The hash table can be thought of as an array on steriods, they are worth reading about, suffice to say
the hash table will tell you when you reach the end of all the entries, and enables us to find entries quickly.

These features efficiently address the addition, removal, and verification of beam parameter sets listed in the above requirements.
*)
{attribute 'reflection'}
FUNCTION_BLOCK FB_Arbiter IMPLEMENTS I_HigherAuthority, I_LowerAuthority
VAR
    nRequestsCount : UDINT; // How many requests are currently in the arbiter

    {attribute 'pytmc' := '
        pv: AP
        io: i
        field: DESC Assertion Pool
     '}
    fbBPAssertionPool    :    FB_BeamParamAssertionPool; //Table of active beam parameter assertions

    xRequestMade : BOOL; // Arbiter has confirmed its request has made it into the beam parameter request

    {attribute 'pytmc' := '
        pv: ArbiterID
        io: i
        field: DESC Arbiter ID for elev. req.
     '}
    nArbiterID : UDINT; // Arbiter ID, used for making higher-level BP requests

    nNextCohort : UDINT := 1; // The cohort ID any new requests will adopt, will become ReqInProgCohort at the start of the next acknowledgement cycle
    nAckInProgCohort : UDINT := 0; // The cohort ID currently being acknowledged, will become nActiveCohort after acknowledgement from HA
    {attribute 'pytmc' := '
        pv: CohortCounter
        io: i
        field: DESC Intrnl cohort counter
     '}
    nActiveCohort : UDINT := 0; // Requests with cohorts <= to this value will be considered active in CheckRequest

    bStartNewAckRequest : BOOL; // Set by an add or remove method call, triggers an ack cycle
    bAckInProgress : BOOL; // Set by ElevateReq when there is a new ack request and reset when the ack cycle is complete

    // The following IDs are set by the last BP request that was most conservative
    // ie. other requests may limit the parameter, but this one is the most recent to limit it
    idTransmission : DWORD; // ID of BP limiting transmission
    idRate : DWORD; // ID of BP limiting rate

    {attribute 'instance-path'}
    {attribute 'noinit'}
    sPath    :    T_MaxString;

    sArbName : T_MaxString;

    InfoStringFmtr : FB_FormatString;

    bVerbose : BOOL := FALSE;
END_VAR
VAR_INPUT
END_VAR
VAR_OUTPUT
    {attribute 'pytmc' := '
        pv: ArbitratedBP
        io: i
        field: DESC Arbitrated BP
     '}
    q_stBeamParams    :    ST_BeamParams := PMPS_GVL.cstFullBeam; //Updated on each cycle of the arbiter FB with the current arbitrated beam parameter set

    q_xStateIDFound    :    BOOL; //Set true if a state-id is found in the assertion pool after calling A_VerifyAssertion
END_VAR

// Adds a request to the arbiter pool.
// Returns true if the request was successfully added, false if not enough space or a request with the same ID is already present.
METHOD AddRequest : BOOL
VAR_INPUT
    nReqID    :    DWORD; // Unique ID within aribter for the request. Make sure this is unique for every device + state combination
    stReqBP        :    ST_BeamParams; //Requested beam params
    sDevName: STRING; // Name of the device making the request
END_VAR
VAR
    BP_Int : ST_BP_ArbInternal;
END_VAR
VAR_INST
    fbLog : FB_LogMessage;
END_VAR
// If the request is already in the pool, then skip the rest.
// This is flawed, needs to update the request if it's already in the pool, despite having the same ID
IF THIS^.CheckRequestInPool(nReqID)
    OR nReqID = PMPS_GVL.EXCLUDED_ASSERTION_ID
    OR nReqID = 0 THEN
    AddRequest := FALSE;
    RETURN;
END_IF


stReqBP.nCohortInt := nNextCohort; // Set the cohort number for this BP request.

// Pack the ID with the request
MEMCPY(ADR(BP_Int), ADR(stReqBP), SIZEOF(stReqBP));
BP_Int.nId := nReqID;
BP_Int.LiveInTable := TRUE;
BP_Int.sDevName := sDevName;

THIS^.fbBPAssertionPool.A_Add(
    key := nReqID,
    putValue := BP_Int
);


IF NOT THIS^.fbBPAssertionPool.bOk THEN
    fbLog(sMsg:=CONCAT('Addition to arbiter assertion pool failed ', DWORD_TO_HEXSTR(nReqID, 4, FALSE)),
            eSevr:=TcEventSeverity.Warning,
            eSubsystem:=E_Subsystem.MPS,
            sJson := F_PMPS_JSON(
                        sArbName,
                        sPath,
                        PMPS_CODES.ARB_FULL));
ELSIF THIS^.fbBPAssertionPool.bOk AND bVerbose THEN
    fbLog(sMsg:=CONCAT('Added to pool ',DWORD_TO_HEXSTR(nReqID, 4, FALSE)),
            eSevr:=TcEventSeverity.Verbose,
            eSubsystem:=E_Subsystem.MPS);
END_IF
// New request, make sure the ack cycle request flag is set
bStartNewAckRequest S= THIS^.fbBPAssertionPool.bOk;

AddRequest := THIS^.fbBPAssertionPool.bOk;

nRequestsCount := nEntryCount;
END_METHOD

// Kernel of the arbiter
// Logic for determining which beam parameter is the most conservative across all request sets.
{attribute 'no_check'}
METHOD INTERNAL ArbitrateBP : ST_BP_ArbInternal
VAR_INPUT
    stBP1    :    ST_BP_ArbInternal;
    stBP2    :    ST_BP_ArbInternal;
END_VAR
VAR
    idx : UINT := 1;
    bcBitmask : WORD:=0;
END_VAR
//<TODO>Add something here to register the key that won for each param

//Attenuation
ArbitrateBP.nTran := MIN(stBP1.nTran, stBP2.nTran);

FOR idx := 1 TO PMPS_GVL.AUX_ATTENUATORS DO
    ArbitrateBP.astAttenuators[idx].nTran := MIN(stBP1.astAttenuators[idx].nTran, stBP2.astAttenuators[idx].nTran);
END_FOR

//Apertures
FOR idx := 1 TO PMPS_GVL.MAX_APERTURES DO
    IF stBP1.astApertures[idx].Height = 0 OR stBP2.astApertures[idx].Height =0 THEN
        ArbitrateBP.astApertures[idx].Height := MAX(stBP1.astApertures[idx].Height, stBP2.astApertures[idx].Height);
    ELSE
        ArbitrateBP.astApertures[idx].Height := MIN(stBP1.astApertures[idx].Height, stBP2.astApertures[idx].Height);
    END_IF

    IF stBP1.astApertures[idx].Width = 0 OR stBP2.astApertures[idx].Width =0 THEN
        ArbitrateBP.astApertures[idx].Width := MAX(stBP1.astApertures[idx].Width, stBP2.astApertures[idx].Width);
    ELSE
        ArbitrateBP.astApertures[idx].Width := MIN(stBP1.astApertures[idx].Width, stBP2.astApertures[idx].Width);
    END_IF
END_FOR

//Photon energy ranges
ArbitrateBP.neVRange := stBP1.neVRange AND stBP2.neVRange;

//Beam Class ranges
ArbitrateBP.nBCRange := stBP1.nBCRange AND stBP2.nBCRange;

//Beam Class
//Assert the highest allowed beamclass
IF (ArbitrateBP.nBCRange = 0) THEN ArbitrateBP.nBeamClass := 0; END_IF
FOR idx:=1 TO 15 BY 1 DO
    IF (idx =1 ) THEN bcBitmask :=1; END_IF
    IF (ArbitrateBP.nBCRange AND bcBitmask) = bcBitmask THEN
        ArbitrateBP.nBeamClass := TO_USINT(idx);
    END_IF
    bcBitmask := ROL(bcBitmask,1);
END_FOR


//Rate
ArbitrateBP.nRate := MIN(stBP1.nRate, stBP2.nRate);
END_METHOD

(* Checks request ID is included in arbitration all the way to the accelerator interface
Use like so:
IF fbArbiter.CheckRequest(nStateIDAssertionToCheck) AND (other logic) THEN:
    Request is found and active in arbitration,. Do something.
ELSE:
    Request was not found, or is not yet included in arbitration. Don't do something/ wait.

*)
METHOD CheckRequest : BOOL
VAR_INPUT
    nReqID    :    DWORD;
END_VAR
VAR
    BP : ST_BeamParams;
END_VAR
fbBPAssertionPool.A_Lookup(key := nReqID);

// Verify BP is acknowledged
BP := fbBPAssertionPool.getValue;

// This logic:
// Did we find the assertion in the pool?
// Is the assertion cohort number less than the current cohort and greater than zero?
// Is the Aribter itself active in arbitration?
CheckRequest := fbBPAssertionPool.bOk AND
                BP.nCohortInt <= nActiveCohort AND
                BP.nCohortInt > 0;
END_METHOD

// Verify request is at least in the local arbiter
// Does not verify request has been included in arbitration.
// Use CheckRequest instead.
METHOD CheckRequestInPool : BOOL
VAR_INPUT
    nReqID    :    DWORD;
END_VAR
THIS^.fbBPAssertionPool.A_Lookup(key := nReqID);

CheckRequestInPool := THIS^.fbBPAssertionPool.bOk;
END_METHOD

// <Arbiter Internal>
// Elevates the arbitrated BP set to something above.
// Could be another arbiter, or a BP requester/ IO,
// or an FB that locks in a specific portion of the BP set.
METHOD ElevateRequest : BOOL
VAR_INPUT
    HigherAuthority : I_HigherAuthority;
END_VAR
(*
This method should only be used with one higher level component.
*)

// Complete previous ack cycle
IF bAckInProgress THEN
    IF HigherAuthority.CheckRequest(nReqID := nArbiterID) THEN
        nActiveCohort := nAckInProgCohort;
        bAckInProgress := FALSE;
    END_IF
END_IF

// Kick off another ack cycle
IF bStartNewAckRequest AND NOT bAckInProgress THEN
    nAckInProgCohort := nNextCohort;
    HigherAuthority.RemoveRequest(nReqID:= nArbiterID);
    bAckInProgress := HigherAuthority.RequestBP(nReqID := nArbiterID, stReqBP := GetArbitratedBP());
    IF bAckInProgress THEN
        bStartNewAckRequest := FALSE;
        nNextCohort := nNextCohort + 1;
    END_IF
END_IF
END_METHOD

METHOD FB_init : BOOL
VAR_INPUT
    bInitRetains : BOOL; // if TRUE, the retain variables are initialized (warm start / cold start)
    bInCopyCode : BOOL;  // if TRUE, the instance afterwards gets moved into the copy code (online change)
    nID : DWORD := PMPS_GVL.EXCLUDED_ASSERTION_ID; // Arbiter ID, must be globally unique cannot be zero or 16#FFFF
END_VAR
nArbiterID := nId;
fbBPAssertionPool.A_Reset();

sArbName := CONCAT('Arbiter ID: 0x', DWORD_TO_HEXSTR(nID, 4, FALSE));
END_METHOD

// Executes Arbitration between all requested beam parameter sets
METHOD INTERNAL GetArbitratedBP : ST_BeamParams
VAR_INPUT
END_VAR
VAR
    getPosPtr    : POINTER TO T_HashTableEntry := 0;
    getBPStructInt    :    ST_BP_ArbInternal;
    stOutputBP    :    ST_BP_ArbInternal; //Holding struct for arbitration process
END_VAR
VAR_INST
    xFirstPass : BOOL := TRUE;
    fbGetCurTaskIdx : GETCURTASKINDEX;
    LastCycleCount : UDINT;
    fbLogMessage : FB_LogMessage;
END_VAR
//Arbitrate
(*
This step cycles through every hash table entry, comparing
the beam parameters from each assertion to what we're planning
to assert.

The safer of the two parameters is kept so at the end we may
have a mix of beam parameters, the composition being safe for
all asserters.

*)

THIS^.fbBPAssertionPool.A_GetFirst( putPosPtr := 0, getPosPtr=>getPosPtr, getValue=>getBPStructInt );
IF THIS^.fbBPAssertionPool.bOk THEN //If the table is empty (not OK), we are left with the default stOutputBP set above.

    //The first entry in the hash table is taken as the setting to arbitrate against
    stOutputBP := getBPStructInt;

    REPEAT
        THIS^.fbBPAssertionPool.A_GetNext( putPosPtr := THIS^.fbBPAssertionPool.getPosPtr, getPosPtr=>getPosPtr, getValue=>getBPStructInt );
        IF THIS^.fbBPAssertionPool.bOk THEN
            stOutputBP := ArbitrateBP(stOutputBP, getBPStructInt);
        END_IF
    UNTIL NOT fbBPAssertionPool.bOk
    END_REPEAT
ELSE
    //Full beam if there are no arbitration requests
    MEMCPY(ADR(stOutputBP), ADR(PMPS_GVL.cstFullBeam), SIZEOF(PMPS_GVL.cstFullBeam));
END_IF

MEMCPY(ADR(q_stBeamParams),ADR(stOutputBP), SIZEOF(q_stBeamParams));

GetArbitratedBP := stOutputBP;

GetArbitratedBP.xValidToggle := NOT GetArbitratedBP.xValidToggle;

xFirstPass := FALSE;
END_METHOD

// How many entries are in the arbiter now
PROPERTY nEntryCount : UDINT
GET
fbBPAssertionPool.A_Count();
IF fbBPAssertionPool.bOk THEN
    nEntryCount := fbBPAssertionPool.nCount ;
END_IF
END_GET
END_PROPERTY

PROPERTY nLowerAuthorityID : DWORD
GET
nLowerAuthorityID := nArbiterID;
END_GET
END_PROPERTY

(* Removes request from abritration. *)
METHOD RemoveRequest : BOOL
VAR_INPUT
    nReqId    :    DWORD;
END_VAR
VAR_INST
    fbLog : FB_LogMessage;
END_VAR
VAR CONSTANT
    BP_Int : ST_BP_ArbInternal := (nId:=0, LiveInTable:=FALSE);
END_VAR
IF nReqId <> PMPS_GVL.EXCLUDED_ASSERTION_ID AND CheckRequestInPool(nReqId) THEN
    // Include an A_Add action here to
    // update this entry with a dummy filler (ID = 0, LiveInTable= False)
    // before removing it since this hash
    // table needs to be viewed with a diagnostic
    // and so the entries need to appear clean.
    THIS^.fbBPAssertionPool.A_Add(key := nReqID, putValue := BP_Int);
    THIS^.fbBPAssertionPool.A_Remove(key := nReqId);

    IF bVerbose THEN
        IF THIS^.fbBPAssertionPool.bOk THEN
                fbLog(sMsg:=CONCAT('Removed from pool: ', DWORD_TO_HEXSTR(nReqID,4,FALSE)),
                eSevr:=TcEventSeverity.Verbose,
                eSubsystem:=E_Subsystem.MPS);
        ELSE
            fbLog(sMsg:=CONCAT('Failed to remove from pool: ', DWORD_TO_HEXSTR(nReqID,4,FALSE)),
                eSevr:=TcEventSeverity.Warning,
                eSubsystem:=E_Subsystem.MPS);
        END_IF
    END_IF

    // With any new request reset the internal arbiter "done" flag
    bStartNewAckRequest S= THIS^.fbBPAssertionPool.bOk;

    RemoveRequest := THIS^.fbBPAssertionPool.bOk;

    nRequestsCount := nEntryCount;

END_IF
END_METHOD

METHOD RequestBP : BOOL
VAR_INPUT
    (*StateID of state requesting beam parameter set*)
    nReqID	: DWORD;
    (*Requested beam params*)
    stReqBP	: ST_BeamParams;
END_VAR
RequestBP := AddRequest(nReqID := nReqID, stReqBP := stReqBP, sDevName:=sArbName);
END_METHOD

END_FUNCTION_BLOCK

// MajorComponents/Arbiter/FB_BeamParamAssertionPool
(* This function block implements simple database. Data element values are stored in the hash table.  *)
{attribute 'no_check'}
FUNCTION_BLOCK FB_BeamParamAssertionPool
VAR_INPUT
    key         : DWORD := 0;(* Entry key: used by A_Lookup, A_Remove method, the key variable is also used by A_Add method *)
    putPosPtr    : POINTER TO T_HashTableEntry := 0;(* Hash table entry position pointer (used by A_Find, A_GetNext, A_GetPrev) *)
    putValue     : ST_BP_ArbInternal;(* Hash table entry value (used by A_AddHead, A_AddTail, A_Find )*)
END_VAR
VAR_OUTPUT
    bOk            : BOOL := FALSE;(* TRUE = Success, FALSE = Failed *)
    getPosPtr    : POINTER TO T_HashTableEntry := 0;(* Returned hash table entry position pointer *)
    getValue     : ST_BP_ArbInternal;(* Returned hash table entry value *)
    nCount        : UDINT := 0;(* Hash table size (number of used entries, used by A_Count) *)
END_VAR
VAR
    {attribute 'pytmc' := '
        pv: Entry
        io: i
     '}
    epicsDataPool    : ARRAY[1..PMPS_PARAM.MAX_ASSERTIONS] OF ST_BP_ArbInternal;(* Structured data element pool for display in EPICS*)
    dataPool    : ARRAY[0..PMPS_PARAM.MAX_ASSERTIONS*3] OF ST_BP_ArbInternal;(* Structured data element pool *)
    entries        : ARRAY[0..PMPS_PARAM.MAX_ASSERTIONS*3] OF T_HashTableEntry;(* Max. number of hash table entries. The value of table entry = 32 bit integer (pointer to dataPool-array-entry) *)
    fbTable     : FB_HashTableCtrl;(* basic hash table control function block *)
    hTable         : T_HHASHTABLE;(* hash table handle *)
    pRefPtr        : POINTER TO ST_BP_ArbInternal := 0;
    indexOfElem    : ULINT;(* Integer value (max. size: x86=>32bit, x64=>64bit)*)
    cstSafeBeam :ST_BeamParams := ( nTran := 0, neVRange := 0, nRate  := 0, nBCRange :=0);// MG
END_VAR

;

ACTION A_Add:
(* Adds entry to the table *)
MEMSET( ADR( getValue ), 0, SIZEOF( getValue ) );
getPosPtr := 0;

fbTable.A_Add( hTable := hTable, key := key, putValue := ADR(cstSafeBeam)(* we will set this value later *), getPosPtr=>getPosPtr, bOk=>bOk );(* Add new element to the table, getPosPtr points to the new entry *)
IF fbTable.bOk THEN(* Success *)
    fbTable.A_GetIndexAtPosPtr( hTable := hTable, putPosPtr := getPosPtr, getValue =>indexOfElem, bOk=>bOk );(* Get array index of getPosPtr entry *)
    IF fbTable.bOk THEN(* Success *)
        pRefPtr     := ADR( dataPool[indexOfElem] );(* Get pointer to the data element *)

        pRefPtr^ := putValue;(* copy application value *)

        fbTable.A_Add( hTable := hTable, key := key, putValue := pRefPtr, bOk=>bOk );(* Assign the entry value = pointer to the data element *)
        IF fbTable.bOk THEN(* Success *)
            getValue := putValue;
        END_IF
    END_IF
END_IF

DataPoolToEpics();
END_ACTION

ACTION A_Count:
(* Count number of used entries *)
nCount := hTable.nCount;
bOk := TRUE;
END_ACTION

ACTION A_GetFirst:
(* Get first entry position pointer and value *)
MEMSET( ADR( getValue ), 0, SIZEOF( getValue ) );
getPosPtr := 0;

fbTable.A_GetFirst( hTable := hTable, putPosPtr := putPosPtr, getValue=>pRefPtr, getPosPtr=>getPosPtr, bOk=>bOk );
IF fbTable.bOk THEN
    getValue := pRefPtr^;
END_IF
END_ACTION

ACTION A_GetNext:
(* Get next entry position pointer and value *)
MEMSET( ADR( getValue ), 0, SIZEOF( getValue ) );
getPosPtr := 0;
bOk := FALSE;

IF putPosPtr = 0 THEN
    RETURN;
END_IF

fbTable.A_GetNext( hTable := hTable, putPosPtr := putPosPtr, getValue=>pRefPtr, getPosPtr=>getPosPtr, bOk=>bOk );
IF fbTable.bOk THEN
    getValue := pRefPtr^;
END_IF
END_ACTION

ACTION A_Lookup:
(* Lookup for entry by key  *)
MEMSET( ADR( getValue ), 0, SIZEOF( getValue ) );
getPosPtr := 0;

fbTable.A_Lookup( key := key, hTable := hTable, putPosPtr := putPosPtr, getValue=>pRefPtr, getPosPtr=>getPosPtr, bOk=>bOk );
IF fbTable.bOk THEN
    getValue := pRefPtr^;
END_IF
END_ACTION

ACTION A_Remove:
(* Search for entry and remove it *)
MEMSET( ADR( getValue ), 0, SIZEOF( getValue ) );
getPosPtr := 0;

fbTable.A_Remove( key := key, hTable := hTable, putPosPtr := putPosPtr, getValue=>pRefPtr, getPosPtr=>getPosPtr, bOk=>bOk );
IF fbTable.bOk THEN
    getValue := pRefPtr^;
END_IF

DataPoolToEpics();
END_ACTION

ACTION A_Reset:
(* Reset/initialize linked list *)
MEMSET( ADR( getValue ), 0, SIZEOF( getValue ) );
getPosPtr := 0;
bOk := F_CreateHashTableHnd( ADR( entries ), SIZEOF( entries ), hTable );(* Intialize table handle *)
fbTable.A_Reset( hTable := hTable, bOk=>bOk );
nCount := 0;
END_ACTION

ACTION DataPoolToEpics:

MEMCPY(ADR(epicsDataPool), ADR(dataPool), (PMPS_PARAM.MAX_ASSERTIONS) * SIZEOF(ST_BP_ArbInternal));
END_ACTION

END_FUNCTION_BLOCK

// MajorComponents/Arbiter/FB_VetoArbiter
FUNCTION_BLOCK FB_VetoArbiter IMPLEMENTS I_HigherAuthority
VAR_INPUT
    bVeto : BOOL := FALSE; // Rising edge clears request, hold true to veto continuously, falling edge restores request
    HigherAuthority : I_HigherAuthority; // Typically connected to a higher-level arbiter.
    LowerAuthority : I_LowerAuthority; // Lower authority to be vetoed
END_VAR
VAR_OUTPUT
END_VAR
VAR_IN_OUT
    FFO : FB_HardwareFFOutput; // This should be the FFO upstream of the veto device
END_VAR
VAR
    ffKeepItSecretKeepItSafe : FB_FastFault := (
        i_xAutoReset := TRUE,
        i_Desc := 'Holds beam off until request is back in arbitration',
        i_TypeCode := 200,
        i_xVetoable := TRUE
    );

    stStandbyBP : ST_BeamParams;


    rtVeto : R_TRIG;
    ftVeto : F_TRIG;
END_VAR


rtVeto(CLK:=bVeto);
ftVeto(CLK:=bVeto);

IF rtVeto.Q THEN
    HigherAuthority.RemoveRequest(LowerAuthority.nLowerAuthorityID);
    HigherAuthority.RequestBP(LowerAuthority.nLowerAuthorityID, PMPS_GVL.cstFullBeam);
ELSIF ftVeto.Q THEN
    HigherAuthority.RemoveRequest(LowerAuthority.nLowerAuthorityID);
    HigherAuthority.RequestBP(LowerAuthority.nLowerAuthorityID, stStandbyBP);
END_IF

LowerAuthority.ElevateRequest(THIS^);

//Fast fault that holds beam off until the request is added back into the system
// when bVeto goes false.
ffKeepItSecretKeepItSafe.i_xOK := HigherAuthority.CheckRequest(LowerAuthority.nLowerAuthorityID) OR bVeto;
ffKeepItSecretKeepItSafe(io_fbFFHWO:=FFO);


METHOD CheckRequest : BOOL
VAR_INPUT
    nReqID	: DWORD;
END_VAR

IF bVeto THEN
    CheckRequest := TRUE;
ELSE
    CheckRequest := HigherAuthority.CheckRequest(nReqID);
END_IF
END_METHOD


METHOD RemoveRequest : BOOL
VAR_INPUT
    (*StateID to remove*)
    nReqID	: DWORD;
END_VAR

IF bVeto THEN
    RemoveRequest := TRUE;
ELSE
    RemoveRequest := HigherAuthority.RemoveRequest(nReqID);
END_IF
END_METHOD

METHOD RequestBP : BOOL
VAR_INPUT
    (*StateID of state requesting beam parameter set*)
    nReqID	: DWORD;
    (*Requested beam params*)
    stReqBP	: ST_BeamParams;
END_VAR

IF NOT bVeto THEN
    // Pass request along to higher authority
    RequestBP := HigherAuthority.RequestBP(nReqID, stReqBP);
ELSE
    RequestBP := TRUE;
END_IF

IF RequestBP THEN
    stStandbyBP := stReqBP;
END_IF
END_METHOD

END_FUNCTION_BLOCK

// MajorComponents/BPTM/BeamParameterTransitionManager
(*
Implements the procedure for safely transitioning between device states.

NOTE:
The BPTM will throw an error if the arbiter does not have enough space for the transition and new final assertion.

 *)
{attribute 'no_check'}
FUNCTION_BLOCK BeamParameterTransitionManager
VAR_IN_OUT

    fbArbiter    :    FB_Arbiter; //Connect to local arbiter

END_VAR
VAR_INPUT
    i_sDeviceName	: 	STRING:='Device'; // Name of the device requesting the transition

    i_TransitionAssertionID    :    UDINT := 0; // Must not be 0 or EXCLUDED_ID
    i_stTransitionAssertion : ST_BeamParams := PMPS_GVL.cst0RateBeam; //Assertion required during transition (always safer than anything inbetween)

    i_nRequestedAssertionID    :    UDINT := 0; // Must not be 0 or EXCLUDED_ID
    i_stRequestedAssertion    :    ST_BeamParams := ( nTran := 0, neVRange := 0, nRate  := 0, nBCRange :=0);// PMPS_GVL.cstSafeBeam; //Requested assertion, change whenever

    i_xMoving    :    BOOL := FALSE; //Provide rising edge when device begins moving <remove>
    i_xDoneMoving    :    BOOL := FALSE; //Provide rising edge when device is done with a move

    stCurrentBeamParameters    :    ST_BeamParams := PMPS_GVL.cstFullBeam; //Connect to current beam parameters

    // Rising edge to cycle back through the BPTM process. Use if something in the process timed out or failed. This will interrupt a current process
    bRetry : BOOL := FALSE;
END_VAR
VAR_OUTPUT

    q_xTransitionAuthorized    :    BOOL := FALSE; //Rising edge indicating the device is safe to move, use as input to move execute (which requires a rising edge)

    bError : BOOL; // Set if some issue occurs within the bptm
    nErrId : UINT; // Set to non-zero to help understand the error.

    bDone : BOOL;
    bBusy : BOOL;

END_VAR

VAR
    nTargetAssertionID    :    UDINT := 0;
    stTargetAssertion    :    ST_BeamParams; // Target assertion
    nCurrentAssertionID    :    UDINT := 0;  // ID of last set state (zero until a state is reached)

    xNewBP    :    BOOL;
    xTranBP    :    BOOL;
    xFinalBPInArb : BOOL;
    xFinalBP    :    BOOL;

    eBPTMState : E_BPTMState := Init;
    ePrevState : E_BPTMState := Init;

    xEntry : BOOL;
    rTransition : R_TRIG;
    xNewTarget : BOOL;

    bTransAssertionFailed : BOOL;
    bFinalAssertionFailed : BOOL;

    LogStrBuffer : ARRAY [0..LogBuffSize] OF STRING;
    LogBuffIdx : FB_Index := (LowerLimit:=0, UpperLimit:=LogBuffSize);

    nAssrtAttempt : INT; // Number of times we have tried asserting a BP set

    rtRetry : R_TRIG;

    rtError : R_TRIG;

    ffTimeout : FB_FastFault := (
        i_Desc := 'Preemptive requests timed out in BPTM',
        i_TypeCode := 16#A,
        i_xAutoReset := FALSE);

    rtDoneMoving : R_TRIG;
    bLatchDoneMoving : BOOL;

    bFirstMove : BOOL := TRUE;

END_VAR
VAR CONSTANT
    LogBuffSize : INT := 40;
    cMaxAttempts : INT := 3;
    (* The thought here is, a BPTM needs at most 2 arbiter slots to complete a transition.
    If we're at capacity, it means some BPTM before this one has begun a transition,
    and will require at least one more arbiter spot to complete.
    *)
    cReqArbCapacity : UDINT := 2;
END_VAR


// Logic for retry button
rtRetry(CLK:=bRetry);
bRetry := FALSE;

// Logic for catching Move Done rising edge
rtDoneMoving(CLK:=i_xDoneMoving);
bLatchDoneMoving S= rtDoneMoving.Q;

// Logic for interrupting BPTM and changing requests
IF nTargetAssertionID <> i_nRequestedAssertionID OR rtRetry.Q THEN

    bError := FALSE;
    nErrID := 0;

    bDone := FALSE;
    bBusy := TRUE;

    // Execute exit actions before transition back to NewTarget
    CASE eBPTMState OF
        Transitioning:
            DeauthorizeTransition();
        //CleaningUp:
    END_CASE

    eBPTMState := E_BPTMState.NewTarget;
    xEntry := eBPTMState <> ePrevState;

END_IF

IF xEntry THEN nAssrtAttempt := 0; END_IF

rtError(CLK:=bError);

IF rtError.Q THEN
    eBPTMState := E_BPTMState.Error;
END_IF

// States
CASE eBPTMState OF
    NewTarget:
        IF xEntry THEN
            NewTarget_ENTRY();
        ELSIF xNewBP THEN
            eBPTMState := E_BPTMState.RequestBP;
        ELSE
            SetNewTarget();
        END_IF

    RequestBP:
        IF PMPS_PARAM.MAX_ASSERTIONS - fbArbiter.nEntryCount >= cReqArbCapacity THEN
            AssertTransitionBP();
            AssertFinalBP();
            eBPTMState := E_BPTMState.WaitForBP;
        ELSE
            LogActions('Arbiter at capacity, leaving space for other BPTM to finish.');
            nErrId := PMPS_CODES.NoRoomInArb;
            bError := TRUE;
        END_IF

    WaitForBP:
        WaitingForTransitionAssertion_DO();
        WaitingForFinalAssertion_DO();
        IF xTranBP AND xFinalBPInArb THEN eBPTMState := E_BPTMState.Transitioning; END_IF

    Transitioning:
        IF xEntry THEN
            AuthorizeTransition();
        ELSIF bLatchDoneMoving OR (bFirstMove AND i_xDoneMoving) THEN
            DeauthorizeTransition();
            eBPTMState := E_BPTMState.WaitForFinalBP;
        END_IF

    WaitForFinalBP:
        xFinalBP := F_SafeBPCompare(stCurrentBeamParameters, stTargetAssertion);
        IF xFinalBP THEN
            eBPTMState := E_BPTMState.CleaningUp;
        END_IF

    CleaningUp:
        IF xEntry THEN
            RemoveTransitionAssertion();
        ELSE
            eBPTMState := E_BPTMState.Done;
        END_IF

    Done:
        bDone := TRUE;
        bFirstMove := FALSE;
        LogActions('Returning to idle');
        eBPTMState := E_BPTMState.Idle;

    Error:
        bError := TRUE;
        eBPTMState := E_BPTMState.Idle;
END_CASE

xEntry := ePrevState <> eBPTMState;
ePrevState := eBPTMState;

bDone R= bError;
bBusy R= bError OR bDone;

ACTION AssertFinalBP:
//q_stFinalAssertion := stTargetAssertion;

//Clearing previous target parameters
(* This is considered safe at this step as the transition
state beam parameters should always be safer than the
current or target state beam parameters
*)
IF nCurrentAssertionID <> 0 THEN
    LogActions(CONCAT('Removing previous request: ', DWORD_TO_HEXSTR(nCurrentAssertionID, 4, false)) );
    fbArbiter.RemoveRequest( nCurrentAssertionID );
END_IF

LogActions(CONCAT('Asserting target req.: ', DWORD_TO_HEXSTR(nTargetAssertionID, 4, false)) );

//Asserting target parameters
bFinalAssertionFailed := NOT fbArbiter.AddRequest(
    nTargetAssertionID,
    stTargetAssertion,
    i_sDeviceName
);

IF bFinalAssertionFailed THEN
    LogActions('Assert final failed. ');
    nAssrtAttempt := nAssrtAttempt + 1;
    IF nAssrtAttempt > cMaxAttempts THEN
        bError := TRUE;
        nErrID := PMPS_CODES.FinalAssrtFail;
    END_IF
ELSE
    // Remembering final assertionID for removal later
    nCurrentAssertionID := nTargetAssertionID;
END_IF
END_ACTION

ACTION AssertTransitionBP:

LogActions( CONCAT('Removing transition id: ', DWORD_TO_STRING(i_TransitionAssertionID)) );
fbArbiter.RemoveRequest(i_TransitionAssertionID);

LogActions( CONCAT('Requesting transition id: ', DWORD_TO_STRING(i_TransitionAssertionID)) );
bTransAssertionFailed := NOT fbArbiter.AddRequest(
    i_TransitionAssertionID,
    i_stTransitionAssertion,
    i_sDeviceName
);

IF bTransAssertionFailed THEN
    LogActions('Assert trans. failed. ');
    nAssrtAttempt := nAssrtAttempt + 1;
    IF nAssrtAttempt > cMaxAttempts THEN
        bError := TRUE;
        nErrID := PMPS_CODES.TransAssrtFail;
    END_IF
END_IF
END_ACTION

ACTION AuthorizeTransition:
q_xTransitionAuthorized := TRUE;

bLatchDoneMoving R= q_xTransitionAuthorized;

LogActions('Authorizing transition');
END_ACTION

ACTION DeauthorizeTransition:
q_xTransitionAuthorized := FALSE;
LogActions('Deauthorizing transition');
END_ACTION

{attribute 'no_check'}
METHOD LogActions : BOOL
VAR_INPUT
    LogStr : STRING;
END_VAR
LogStrBuffer[LogBuffIdx.IncVal()] := LogStr;
END_METHOD

ACTION NewTarget_ENTRY:
xNewBP := False;
END_ACTION

ACTION RemoveTransitionAssertion:
//q_stTransitionAssertion := PMPS_GVL.cstFullBeam;

//Removing transition assertion
fbArbiter.RemoveRequest( i_TransitionAssertionID );

LogActions('Removing transition req');

//TODO add something to verify removal
END_ACTION

ACTION RequestBP_DO:
// Request BP atomically so we know we'll finish the BPTM cycle
IF fbArbiter.nEntryCount < cReqArbCapacity THEN

    LogActions( CONCAT('Removing transition id: ', DWORD_TO_STRING(i_TransitionAssertionID)) );
    fbArbiter.RemoveRequest(i_TransitionAssertionID);

    LogActions( CONCAT('Requesting transition id: ', DWORD_TO_STRING(i_TransitionAssertionID)) );
    bTransAssertionFailed := NOT fbArbiter.AddRequest(
        i_TransitionAssertionID,
        i_stTransitionAssertion,
        i_sDeviceName
    );

    IF bTransAssertionFailed THEN
        LogActions('Assert trans. failed. ');
        nAssrtAttempt := nAssrtAttempt + 1;
        IF nAssrtAttempt > cMaxAttempts THEN
            bError := TRUE;
            nErrID := PMPS_CODES.TransAssrtFail;
        END_IF
    END_IF



ELSE
    LogActions('Arbiter at capacity, leaving space for other BPTM to finish.');
END_IF
END_ACTION

ACTION SetNewTarget:

IF F_ValidReqID(i_nRequestedAssertionID) AND
    F_ValidReqID(i_TransitionAssertionID) THEN

    stTargetAssertion := i_stRequestedAssertion;
    nTargetAssertionID := i_nRequestedAssertionID;

    LogActions('New target set');

    xNewBP := TRUE;

ELSE
    IF NOT F_ValidReqID(i_nRequestedAssertionID) THEN

        nErrID := PMPS_CODES.BadTargetID;
    ELSIF NOT F_ValidReqID(i_TransitionAssertionID) THEN
        nErrID := PMPS_CODES.BadTransID;
    END_IF
    LogActions('Error in set new target');
    bError := TRUE;
END_IF
END_ACTION

ACTION WaitingForFinalAssertion_DO:
//Final Assertion Verification

xFinalBPInArb := fbArbiter.CheckRequest( i_nRequestedAssertionID);;
END_ACTION

ACTION WaitingForFinalAssertion_EXIT:
//Set this bool false so we can get a rising edge on the next try
xFinalBP := FALSE;
END_ACTION

ACTION WaitingForTransitionAssertion_DO:
//Transition Assertion Verification
xTranBP    := F_SafeBPCompare0Rate(stCurrentBeamParameters, i_stTransitionAssertion) AND
    fbArbiter.CheckRequest(i_TransitionAssertionID);
END_ACTION

ACTION WaitingForTransitionAssertion_EXIT:
xTranBP := FALSE;
END_ACTION

END_FUNCTION_BLOCK

// MajorComponents/InterPlcComm/FB_ArbiterToSubSys_IO
(* Exchanges preemption requests and current beam state with subsystems in arbiter
network.

2019-12-2, A. Wallace

Use in conjunction with FB_SubSysToArbiter_IO.

This FB runs in the beamline arbiter PLC (BAP). There should be one of these for every
subsystem interfaced to the BAP. Each subsystem PLC should run a sibling FB_SubSysToArbiter_IO FB.

This FB and its subordinate communicate through the ethercat connection between the subsystem PLC and the BAP.

A beam parameter set request is sent from the subsystem to this PLC, and includes a cohort number.

This cohort number (i_RequestedBP.nCohortInt) is compared to a local cohort number (nRequestedCohort).
A request from the subsystem to update or modify its current request is indicated by an increase in the
i_RequestedBP.nCohortInt value. Then this function block updates the local arbiter request for the subsystem
and awaits confirmation. Once the new request is confirmed in the preemptive system this function block increments
the ActiveCohort value to match the nRequestedCohort. ActiveCohort is also relayed back to the subsystem
as the active cohort value in the o_CurrentBP set. The subsystem then knows its request has been heard,
and can carry out its own acknowledgement to its various requestors.

Things to note:
If a subsystem has any new or changed preemptive requests you should see the cohort value increment a bit.
If the cohort number is incrementing out of control, it usually means the subsysetm has some preemptive
request loop (two arbiters elevating to each other), or there is a RequestAdd, RequestRemove loop.

*)
FUNCTION_BLOCK FB_ArbiterToSubSys_IO
VAR_INPUT
    RequestingSystemID	:	DWORD := PMPS_GVL.EXCLUDED_ASSERTION_ID; // System ID for making requests to the supreme arbiter
    sName : STRING := 'ArbiterToSubSys';
    Reset : BOOL;
END_VAR
VAR_OUTPUT
END_VAR
VAR_IN_OUT
    Arbiter	: FB_Arbiter;
    fbFFHWO : FB_HardwareFFOutput;
END_VAR
VAR

    i_RequestedBP AT %I*	:	ST_BeamParams_IO; // Requested BP from subsystem
    {attribute 'pytmc' := '
        pv: RequestedBP:FromSubSys
    '}
    RequestedBP: ST_BeamParams;

    o_CurrentBP AT %Q* : ST_BeamParams_IO; // Current BP set

    // EL6692 Diagnostics
    i_Connected AT %I* : BOOL; // SYNC Inputs^External device not connected !!! Doesn't really work.
    {attribute 'pytmc' := 'pv: WcState
        io: i
        field: DESC Working counter state.
        field: ZNAM OK
        field: ONAM Error'}
    i_WcState AT %I* : BOOL := TRUE; // WcState^WcState
    {attribute 'pytmc' := 'pv: TxPDO_state
        io: i
        field: DESC PDO Transmission is OK
        field: ZNAM OK
        field: ONAM Error'}
    i_TxPDOState AT %I* : BOOL := TRUE; // SYNC Inputs^TxPDO state
    {attribute 'pytmc' := 'pv: TxPDO_toggle
        io: i
        field: DESC PDO Transmission is OK
        field: ZNAM OK
        field: ONAM Error'}
    i_TxPDOToggle AT %I* : BOOL; // TxPDO toggle

    // Fast faults
    ffPMPSIO_Disconnect : FB_FastFault := (i_Desc:='Issue w/ arbiter interface to subsystem, verify subsystem is OK, or ethercat connection.'); // Fast fault for ethercat issues
    nActiveCohort : UDINT := 0; // Active cohort. Updated to the req. number from the sub system after request is confirmed.
    nRequestedCohort : UDINT := 0;
    rtToggle : R_TRIG;


END_VAR


// Incoming request from subsystem PLC
RequestedBP := IO_TO_BP(i_RequestedBP);

// Update Arbiter with our request
rtToggle(CLK:= i_RequestedBP.xValid); // If interface resumes, reset/catch up
// xValid will go false if the PLC program on the other side is stopped. Ironically the ethercat interface continues happily.
// If subsystem cohort has incremented, update beam parameter request with our arbiter
IF rtToggle.Q THEN
    nActiveCohort := 0;
END_IF

IF i_RequestedBP.nCohortInt > nRequestedCohort OR rtToggle.Q THEN
    Arbiter.RemoveRequest(RequestingSystemID);
    Arbiter.AddRequest(RequestingSystemID, RequestedBP,sName);
    nRequestedCohort := i_RequestedBP.nCohortInt;
END_IF


// Check if latest request is acknowledged by this arbiter
// Acknowledgement happens after an arbitration cycle, which means if RequestedCohort just incremented
// due to a new request, CheckRequest will be false.
IF Arbiter.CheckRequest(RequestingSystemID) THEN
    nActiveCohort := nRequestedCohort; // If it is, then the active cohort is set to the requested cohort number.
END_IF

// Sending current beam parameter set to subsystems
o_CurrentBP := BP_TO_IO(PMPS_GVL.stCurrentBeamParameters);
o_CurrentBP.nCohortInt := nActiveCohort;


//////////////////////////////////////
// Verifying the ethercat interface health
/////////////////////////////////////
// Both of these values should be 0 for a fully valid exchange
ffPMPSIO_Disconnect.i_xOK := NOT i_WcState AND NOT i_TxPDOState;

ffPMPSIO_Disconnect(
    io_fbFFHWO := fbFFHWO,
    i_xReset := Reset,
    i_DevName := sName,
    i_TypeCode:=5);

END_FUNCTION_BLOCK

// MajorComponents/InterPlcComm/FB_SubSysToArbiter_IO
// Use on a subsystem PLC to request from the arbiter
// Run at the top of your cycle to receive the latest BP
FUNCTION_BLOCK FB_SubSysToArbiter_IO IMPLEMENTS I_HigherAuthority
VAR_INPUT
    Reset : BOOL; // Fast fault reset
    sName : STRING := 'SubSysToArbiter';
    i_bVeto : BOOL;
END_VAR
VAR_OUTPUT
END_VAR
VAR_IN_OUT
    Arbiter	: FB_Arbiter;
    fbFFHWO : FB_HardwareFFOutput;
END_VAR
VAR
    {attribute 'TcLinkTo' := 'TIIB[PMPS_PRE]^IO Inputs^CurrentBP'}
    i_stCurrentBP    AT %I* :    ST_BeamParams_IO;
    {attribute 'TcLinkTo' := 'TIIB[PMPS_PRE]^IO Outputs^RequestedBP'}
    q_stRequestedBP AT %Q* :    ST_BeamParams_IO;
    {attribute 'pytmc' := 'pv: TxPDO_toggle
        io: i'}
    {attribute 'TcLinkTo' := 'TIIB[PMPS_PRE]^SYNC Inputs^TxPDO toggle'}
    xTxPDO_toggle    AT     %I* :    BIT;
    {attribute 'pytmc' := 'pv: TxPDO_state
        io: i'}
    {attribute 'TcLinkTo' := 'TIIB[PMPS_PRE]^SYNC Inputs^TxPDO state'}
    xTxPDO_state    AT    %I*    :    BIT;


    // Fast faults
    ffPMPSIO_Disconnect : FB_FastFault := (i_Desc:='Arbiter network interface disconnected or not OP',i_DevName := sName);

    // A request is not considered included until the active cohort number is >= the request cohort number.
    {attribute 'pytmc' := 'pv: RequestCohort
        io: i'}
    nRequestCohort : UDINT := 0; // Request cohort
    {attribute 'pytmc' := 'pv: ActiveCohort
        io: i'}
    nActiveCohort : UDINT := 0; // Active cohort, updated by incoming BP from arbiter PLC, in the ElevateRequest arbiter call

    fbVetoArb : FB_VetoArbiter;

    fbLog : FB_LogMessage;
END_VAR

//Receiving current BP state
PMPS_GVL.stCurrentBeamParameters := IO_TO_BP(i_stCurrentBP);
PMPS_GVL.stCurrentBeamParameters.xValidToggle := xTxPDO_toggle; // This line must follow the one above. Sequence is important.

// Forwarding BP request for the subsystem
fbVetoArb.bVeto := i_bVeto;
fbVetoArb(HigherAuthority:=THIS^, LowerAuthority:=Arbiter, FFO:=fbFFHWO);

//Broadcasting current request
PMPS_GVL.stRequestedBeamParameters := IO_TO_BP(q_stRequestedBP);


q_stRequestedBP.xValid := TRUE; // This is set and held true here every cycle to prove the PLC on this side is still running

ffPMPSIO_Disconnect(
    i_xOK := xTxPDO_state = 0,
    io_fbFFHWO := fbFFHWO,
    i_xReset := Reset,
    i_DevName := sName,
    i_TypeCode := 6,
    i_xVetoable := FALSE
    );

METHOD CheckRequest : BOOL
VAR_INPUT
    nReqID	: DWORD;
END_VAR
VAR_INST
    xFirstTime : BOOL := TRUE;
    nId : DWORD;
END_VAR
// Check this id matches what we've seen before
IF xFirstTime THEN
    nId := nReqId;
ELSIF nId <> nReqId THEN
    fbLog(sMsg := 'SubSysToArbiter Check mismatched with a different ID', eSevr := TcEventSeverity.Error);
    RETURN;
END_IF

nActiveCohort := ULINT_TO_UDINT(i_stCurrentBP.nCohortInt);

// i_stCurrentBP.nCohortInt is incremented by the FB_ArbiterToSubSys block on the other side of the EL669* interface
CheckRequest := nRequestCohort <= nActiveCohort;
END_METHOD

METHOD RemoveRequest : BOOL
VAR_INPUT
    nReqID    :    DWORD; //StateID to remove
END_VAR
// Update internal BP request struct
q_stRequestedBP := BP_TO_IO(PMPS_GVL.cstFullBeam);

nRequestCohort := nRequestCohort + 1;

// Mark the current cohort id
q_stRequestedBP.nCohortInt := nRequestCohort;

RemoveRequest := TRUE;
END_METHOD

METHOD RequestBP : BOOL
VAR_INPUT
    (*StateID of state requesting beam parameter set*)
    nReqID	: DWORD;
    (*Requested beam params*)
    stReqBP	: ST_BeamParams;
END_VAR
// Check the request is coming from the same source we're used to

// Update internal BP request struct
q_stRequestedBP := BP_TO_IO(stReqBP);

nRequestCohort := nRequestCohort + 1;

// Mark the current cohort id
q_stRequestedBP.nCohortInt := nRequestCohort;

RequestBP := TRUE;
END_METHOD

END_FUNCTION_BLOCK

// MajorComponents/PhotonEnergyInterface/F_CalculatePhotonEnergy
FUNCTION F_CalculatePhotonEnergy : LREAL
VAR_INPUT
    (* Electron energy in GeV *)
    fElectronEnergy_GeV : LREAL;
    (* Undulator period in mm *)
    fUndulatorPeriod_mm : LREAL;
    (* Unitless undulator K parameter / strength *)
    fUndulatorStrength : LREAL;
END_VAR

VAR
    fDenominator: LREAL;
END_VAR

VAR CONSTANT
    (* GeV [electron rest mass/energy] *)
    m_e : LREAL := 0.0005109989461;
    (* Js [Planck's constant] *)
    h 	: LREAL := 6.62607004E-34;
    (* C [electron charge] *)
    e 	: LREAL := 1.6021766208E-19;
    (* m/s, speed of light *)
    c 	: LREAL := 299792458;

END_VAR

(*

Reference Python implementation

def calculate_photon_energy(electron_energy, period, k):
    '''
    Calculate photon energy, in eV.

    Parameters
    ----------
    electron_energy : float
        Electron energy in GeV

    period : float
        Undulator period, in mm

    k : float
        Undulator K parameter (strength), unitless
    '''
    m_e = 0.0005109989461  # GeV [electron rest mass/energy]
    h = 6.62607004e-34  # Js [Planck's constant]
    e = 1.6021766208e-19  # C [electron charge]
    c = 299792458  # m/s, speed of light
    return ((2. * (electron_energy / m_e) ** 2 * h * c) /
            (e * period * 1e-3 * (1 + k ** 2 / 2.)))

*)
fDenominator := (e * fUndulatorPeriod_mm * 1E-3 * (1.0 + EXPT(fUndulatorStrength, 2.0) / 2.0));
F_CalculatePhotonEnergy := (2.0 * EXPT(fElectronEnergy_GeV / m_e, 2.0) * h * c) / MAX(fDenominator, 4.94065645841247E-324);

END_FUNCTION

// MajorComponents/PhotonEnergyInterface/FB_AcceleratorLinks
FUNCTION_BLOCK FB_AcceleratorLinks
VAR_INPUT

END_VAR

VAR_OUTPUT
END_VAR


VAR

    {attribute 'pytmc' := '
        pv: eEnrg:Hgvpu
        link: BEND:DMPH:400:BACT
        field: EGU GeV
    '}
    fbHgvpuElectronEnergy : FB_LREALFromEPICS;

    {attribute 'pytmc' := '
        pv: eEnrg:SXU
        link: BEND:DMPS:400:BACT
        field: EGU GeV
    '}
    fbSxuElectronEnergy : FB_LREALFromEPICS;

END_VAR

fbHgvpuElectronEnergy();
fbSxuElectronEnergy();

END_FUNCTION_BLOCK

// MajorComponents/PhotonEnergyInterface/FB_Hgvpu
FUNCTION_BLOCK FB_Hgvpu IMPLEMENTS I_UndulatorComplex
VAR_INPUT
    fbElectronEnergy : REFERENCE TO FB_LREALFromEPICS;
END_VAR

VAR_OUTPUT
    {attribute 'pytmc' := '
        pv: CurrentPhotonEnergy
        io: i
        field: DESC Calculated current photon energy
        field: PREC 3
        field: EGU eV
    '}
    fCurrentPhotonEnergy : LREAL;
    {attribute 'pytmc' := '
        pv: TargetPhotonEnergy
        io: i
        field: DESC Calculated desired photon energy
        field: PREC 3
        field: EGU eV
    '}
    fTargetPhotonEnergy : LREAL;
    {attribute 'pytmc' := '
        pv: SeedUndulatorNumber
        io: i
        field: DESC Seed undulator number
    '}
    nSeedUndulator : UDINT; // Set to zero when no undulators are active
    {attribute 'pytmc' := '
        pv: TargetSeedUndulatorNumber
        io: i
        field: DESC Seed undulator number for target K
    '}
    nTargetSeedUndulator : UDINT; // Set to zero when no undulators are active
END_VAR


VAR
    // From lcls-srv01: grep -e KDes  /u1/lcls/epics/ioc/data/ioc-undh-uc*/iocInfo/IOC.pvlist |sort

    {attribute 'pytmc' := 'pv: 24; link: 2450:'}
    fbSegment_24 : FB_UndulatorSegment;

    {attribute 'pytmc' := 'pv: 25; link: 2550:'}
    fbSegment_25 : FB_UndulatorSegment;

    {attribute 'pytmc' := 'pv: 26; link: 2650:'}
    fbSegment_26 : FB_UndulatorSegment;

    {attribute 'pytmc' := 'pv: 27; link: 2750:'}
    fbSegment_27 : FB_UndulatorSegment;

    {attribute 'pytmc' := 'pv: 29; link: 2950:'}
    fbSegment_29 : FB_UndulatorSegment;

    {attribute 'pytmc' := 'pv: 30; link: 3050:'}
    fbSegment_30 : FB_UndulatorSegment;

    {attribute 'pytmc' := 'pv: 31; link: 3150:'}
    fbSegment_31 : FB_UndulatorSegment;

    {attribute 'pytmc' := 'pv: 32; link: 3250:'}
    fbSegment_32 : FB_UndulatorSegment;

    {attribute 'pytmc' := 'pv: 33; link: 3350:'}
    fbSegment_33 : FB_UndulatorSegment;

    {attribute 'pytmc' := 'pv: 34; link: 3450:'}
    fbSegment_34 : FB_UndulatorSegment;

    {attribute 'pytmc' := 'pv: 35; link: 3550:'}
    fbSegment_35 : FB_UndulatorSegment;

    {attribute 'pytmc' := 'pv: 36; link: 3650:'}
    fbSegment_36 : FB_UndulatorSegment;

    {attribute 'pytmc' := 'pv: 37; link: 3750:'}
    fbSegment_37 : FB_UndulatorSegment;

    {attribute 'pytmc' := 'pv: 38; link: 3850:'}
    fbSegment_38 : FB_UndulatorSegment;

    {attribute 'pytmc' := 'pv: 39; link: 3950:'}
    fbSegment_39 : FB_UndulatorSegment;

    {attribute 'pytmc' := 'pv: 40; link: 4050:'}
    fbSegment_40 : FB_UndulatorSegment;

    {attribute 'pytmc' := 'pv: 41; link: 4150:'}
    fbSegment_41 : FB_UndulatorSegment;

    {attribute 'pytmc' := 'pv: 42; link: 4250:'}
    fbSegment_42 : FB_UndulatorSegment;

    {attribute 'pytmc' := 'pv: 43; link: 4350:'}
    fbSegment_43 : FB_UndulatorSegment;

    {attribute 'pytmc' := 'pv: 44; link: 4450:'}
    fbSegment_44 : FB_UndulatorSegment;

    {attribute 'pytmc' := 'pv: 45; link: 4550:'}
    fbSegment_45 : FB_UndulatorSegment;

    {attribute 'pytmc' := 'pv: 46; link: 4650:'}
    fbSegment_46 : FB_UndulatorSegment;

    fbSegment : ARRAY [iLowBound_LUnd..iHighBound_LUnd] OF POINTER TO FB_UndulatorSegment;
    fbCurrentSegment : REFERENCE TO FB_UndulatorSegment;

    iIndex : UDINT;

    bInitialized : BOOL := FALSE;

END_VAR

VAR CONSTANT
    {attribute 'pytmc' := '
        pv: FirstSegment
        io: i
    '}
    iLowBound_LUnd  : UDINT := 24;

    {attribute 'pytmc' := '
        pv: LastSegment
        io: i
    '}
    iHighBound_LUnd : UDINT := 46;

    {attribute 'pytmc' := '
        pv: Period
        io: i
        field: EGU mm
    '}
    fPeriod_mm_LUnd : LREAL := 26.0;

    {attribute 'pytmc' := '
        pv: LowK
        io: i
    '}
    fLowK_LUnd : LREAL := 0.54;

    {attribute 'pytmc' := '
        pv: HiK
        io: i
    '}
    fHiK_LUnd : LREAL := 2.6;
END_VAR

IF NOT bInitialized THEN
    Init();
END_IF

UndAdrUpdate();

nSeedUndulator := 0;
nTargetSeedUndulator := 0;

FOR iIndex := iLowBound_LUnd TO iHighBound_LUnd DO
    IF fbSegment[iIndex] <> 0 THEN
        fbCurrentSegment REF= fbSegment[iIndex]^;
        fbCurrentSegment(fbElectronEnergy:=fbElectronEnergy);

        //Mark the seed undulator, first undulator operating within K bounds
        IF fbCurrentSegment.xActive AND nSeedUndulator = 0 THEN
            nSeedUndulator := iIndex;
            fCurrentPhotonEnergy := fbCurrentSegment.fPhotonEnergyAct;
        END_IF

        IF fbCurrentSegment.xTargetActive AND nTargetSeedUndulator = 0 THEN
            nTargetSeedUndulator := iIndex;
            fTargetPhotonEnergy := fbCurrentSegment.fPhotonEnergyDes;
        END_IF
    END_IF
END_FOR

IF nSeedUndulator = 0 THEN
    fCurrentPhotonEnergy := 0;
END_IF

IF nTargetSeedUndulator = 0 THEN
    fTargetPhotonEnergy := 0;
END_IF

ACTION Init:

UndAdrUpdate();


    FOR iIndex := iLowBound_LUnd TO iHighBound_LUnd DO
            IF fbSegment[iIndex] <> 0 THEN
            fbCurrentSegment REF= fbSegment[iIndex]^;
            fbCurrentSegment.fPeriod_mm := fPeriod_mm_LUnd;
            fbCurrentSegment.fLowK := fLowK_LUnd;
            fbCurrentSegment.fHiK := fHiK_LUnd;
        END_IF
    END_FOR

    bInitialized := TRUE;
END_ACTION

PROPERTY rCurrentPhotonEnergy : REAL
GET
rCurrentPhotonEnergy := fCurrentPhotonEnergy;
END_GET
END_PROPERTY

PROPERTY rTargetPhotonEnergy : REAL
GET
rTargetPhotonEnergy := fTargetPhotonEnergy;
END_GET
END_PROPERTY

ACTION UndAdrUpdate:
fbSegment[24] := ADR(fbSegment_24);
fbSegment[25] := ADR(fbSegment_25);
fbSegment[26] := ADR(fbSegment_26);
fbSegment[27] := ADR(fbSegment_27);
fbSegment[28] := 0;
fbSegment[29] := ADR(fbSegment_29);
fbSegment[30] := ADR(fbSegment_30);
fbSegment[31] := ADR(fbSegment_31);
fbSegment[32] := ADR(fbSegment_32);
fbSegment[33] := ADR(fbSegment_33);
fbSegment[34] := ADR(fbSegment_34);
fbSegment[35] := ADR(fbSegment_35);
fbSegment[36] := ADR(fbSegment_36);
fbSegment[37] := ADR(fbSegment_37);
fbSegment[38] := ADR(fbSegment_38);
fbSegment[39] := ADR(fbSegment_39);
fbSegment[40] := ADR(fbSegment_40);
fbSegment[41] := ADR(fbSegment_41);
fbSegment[42] := ADR(fbSegment_42);
fbSegment[43] := ADR(fbSegment_43);
fbSegment[44] := ADR(fbSegment_44);
fbSegment[45] := ADR(fbSegment_45);
fbSegment[46] := ADR(fbSegment_46);
END_ACTION

END_FUNCTION_BLOCK

// MajorComponents/I_UndulatorComplex
INTERFACE I_UndulatorComplex

PROPERTY rCurrentPhotonEnergy : REAL
GET
END_GET
END_PROPERTY

PROPERTY rTargetPhotonEnergy : REAL
GET
END_GET
END_PROPERTY

END_INTERFACE

// MajorComponents/PhotonEnergyInterface/FB_UndulatorSegment
FUNCTION_BLOCK FB_UndulatorSegment
VAR_INPUT	
	(* Undulator period in millimeters, to be set by subclasses for HXR, read by pv for SXR, left here for backward compatability *)
    fPeriod_mm : LREAL := 1.0;
	
    fbElectronEnergy : REFERENCE TO FB_LREALFromEPICS;

    fLowK : LREAL := 0;
    fHiK : LREAL := 6;
    fKRangeHyst : LREAL := 0.01;
END_VAR

VAR_OUTPUT
    {attribute 'pytmc' := '
        pv: eVAct
        field: DESC Calculated photon energy
        field: PREC 3
        field: EGU eV
    '}
    fPhotonEnergyAct : LREAL;

    {attribute 'pytmc' := '
        pv: eVDes
        field: DESC Calculated desired photon energy
        field: PREC 3
        field: EGU eV
    '}
    fPhotonEnergyDes : LREAL;

    {attribute 'pytmc' := '
        pv: Active
        io: i
        field: DESC Undulator is considered active
    '}
    xActive : BOOL; // Undulator is considered active

    {attribute 'pytmc' := '
        pv: TargetActive
        io: i
        field: DESC Target K would make und active
    '}
    xTargetActive : BOOL; // Undulator is considered active at this target

    {attribute 'pytmc' := '
        pv: KAct
        io: i
        field: DESC Current K
    '}
    fKAct : LREAL;

    {attribute 'pytmc' := '
        pv: KDes
        io: i
        field: DESC Target K
    '}
    fKDes : LREAL;
	
	{attribute 'pytmc' := '
        pv: Lambda_U
        io: i
        field: DESC Period in m
    '}
    fLambda_U : LREAL;

    {attribute 'pytmc' := '
        pv: KActValid
        io: i
        field: DESC Current K Readback Valid
    '}
    bKActValid : BOOL;

    {attribute 'pytmc' := '
        pv: KDesValid
        io: i
        field: DESC Target K Readback Valid
    '}
    bKDesValid : BOOL;
	
	 {attribute 'pytmc' := '
        pv: lambdaValid
        io: i
        field: DESC lambda_U Readback Valid
    '}
    blambdaValid : BOOL;


END_VAR

VAR
    {attribute 'pytmc' := '
        pv: KDes
        link: KDes
    '}
    fbKDesired : FB_LREALFromEPICS;

    {attribute 'pytmc' := '
        pv: KAct
        link: KAct
    '}
    fbKActual : FB_LREALFromEPICS;
	
	{attribute 'pytmc' := '
        pv: lambda_U
        link: lambda_U
    '}
    fblambda_U : FB_LREALFromEPICS;

END_VAR

fbKDesired();
fbKActual();
fblambda_U();

fKAct := fbKActual.fValue;
bKActValid := fbKActual.bValid;
fKDes := fbKDesired.fValue;
bKDesValid := fbKDesired.bvalid;
fLambda_U := fblambda_U.fValue;
blambdaValid:= fblambda_U.bValid;

IF __ISVALIDREF(fbElectronEnergy) THEN

    IF fbKActual.bValid AND fblambda_U.bValid AND fbElectronEnergy.bValid THEN
        fPhotonEnergyAct := F_CalculatePhotonEnergy(
            fElectronEnergy_GeV:=fbElectronEnergy.fValue,
            fUndulatorPeriod_mm:=fPeriod_mm,
            fUndulatorStrength:=fbKActual.fValue
        );

        //Set this undulator active if actual K is within operational range
        xActive S= fLowK <= fbKActual.fValue AND fbKActual.fValue <= fHiK AND
        (fbKActual.bValid AND fbKActual.bValid);
        xActive R= (fLowK - fKRangeHyst) > fbKActual.fValue OR fbKActual.fValue > (fHiK + fKRangeHyst) OR
                    (NOT fbKActual.bValid OR NOT fbKActual.bValid);

        //Set this undulator active if target K is within operational range
        xTargetActive S= fLowK <= fbKDesired.fValue AND fbKDesired.fValue <= fHiK AND
        (fbKDesired.bValid AND fbKDesired.bValid);
        xTargetActive R= (fLowK - fKRangeHyst) > fbKDesired.fValue OR fbKDesired.fValue > (fHiK + fKRangeHyst) OR
                    (NOT fbKDesired.bValid OR NOT fbKDesired.bValid);
    END_IF

    IF fbKDesired.bValid AND fblambda_U.bValid AND fbElectronEnergy.bValid THEN
        fPhotonEnergyDes := F_CalculatePhotonEnergy(
            fElectronEnergy_GeV:=fbElectronEnergy.fValue,
            fUndulatorPeriod_mm:=fPeriod_mm,
            fUndulatorStrength:=fbKDesired.fValue
        );
    END_IF

END_IF

END_FUNCTION_BLOCK

// MajorComponents/PhotonEnergyInterface/FB_KPhotonEnergy
FUNCTION_BLOCK FB_KPhotonEnergy EXTENDS FB_PhotonEnergy
VAR_INPUT
END_VAR
VAR_OUTPUT
END_VAR
VAR
    {attribute 'pytmc' := '
        pv: eEnrg
        link: BEND:DMPS:400:BACT
        field: EGU GeV
    '}
    fbSxuElectronEnergy : FB_LREALFromEPICS;

    {attribute 'pytmc' := '
        pv: EEnergy
        io: i
        field: DESC Electron Energy
        field: EGU GeV
    '}
    fElectronEnergyVal : LREAL;

    {attribute 'pytmc' := '
        pv: EEnergyValid
        io: i
        field: DESC Electron Energy Valid
    '}
    bElectronEnergyValid : BOOL;

    {attribute 'pytmc' := '
        pv: UND
        link: USEG:UNDS:
    '}
    fbSxu : FB_SXU;

END_VAR

// Update PVs
fbSxuElectronEnergy();

fElectronEnergyVal := fbSxuElectronEnergy.fValue;
bElectronEnergyValid := fbSxuElectronEnergy.bValid;

fbSxu(fbElectronEnergy:=fbSxuElectronEnergy);

SUPER^(BP:=SUPER^.BP, Undulator:=fbSxu );

END_FUNCTION_BLOCK

// MajorComponents/PhotonEnergyInterface/FB_PhotonEnergy
FUNCTION_BLOCK FB_PhotonEnergy
VAR_INPUT
    Undulator : I_UndulatorComplex;
END_VAR
VAR_OUTPUT
END_VAR
VAR_IN_OUT
    BP : ST_BeamParams;
END_VAR
VAR
    nCurrentPhotonEnergyBitmask : UDINT;
    nTargetPhotonEnergyBitmask : UDINT;
END_VAR


//Update BP
nCurrentPhotonEnergyBitmask := F_eVRangeCalculator(Undulator.rCurrentPhotonEnergy, nCurrentPhotonEnergyBitmask);
nTargetPhotonEnergyBitmask := F_eVRangeCalculator(Undulator.rTargetPhotonEnergy, nTargetPhotonEnergyBitmask);

BP.neVRange := nCurrentPhotonEnergyBitmask OR nTargetPhotonEnergyBitmask;

END_FUNCTION_BLOCK

// MajorComponents/PhotonEnergyInterface/FB_SXU
FUNCTION_BLOCK FB_SXU IMPLEMENTS I_UndulatorComplex
VAR_INPUT
    fbElectronEnergy : REFERENCE TO FB_LREALFromEPICS;
END_VAR

VAR_OUTPUT
    {attribute 'pytmc' := '
        pv: CurrentPhotonEnergy
        io: i
        field: DESC Calculated current photon energy
        field: PREC 3
        field: EGU eV
    '}
    fCurrentPhotonEnergy : LREAL;
    {attribute 'pytmc' := '
        pv: TargetPhotonEnergy
        io: i
        field: DESC Calculated desired photon energy
        field: PREC 3
        field: EGU eV
    '}
    fTargetPhotonEnergy : LREAL;
        {attribute 'pytmc' := '
        pv: SeedUndulatorNumber
        io: i
        field: DESC Seed undulator number
    '}
    nSeedUndulator : UDINT; // Set to zero when no undulators are active
    {attribute 'pytmc' := '
        pv: TargetSeedUndulatorNumber
        io: i
        field: DESC Seed undulator number for target K
    '}
    nTargetSeedUndulator : UDINT; // Set to zero when no undulators are active
END_VAR



VAR
    // From lcls-srv01: grep -e KDes  /u1/lcls/epics/ioc/data/sioc-unds-uc*/iocInfo/IOC.pvlist |sort

    {attribute 'pytmc' := 'pv: 21; link: 2150:'}
    fbSegment_21 : FB_UndulatorSegment;

    {attribute 'pytmc' := 'pv: 22; link: 2250:'}
    fbSegment_22 : FB_UndulatorSegment;

    {attribute 'pytmc' := 'pv: 23; link: 2350:'}
    fbSegment_23 : FB_UndulatorSegment;

    {attribute 'pytmc' := 'pv: 24; link: 2450:'}
    fbSegment_24 : FB_UndulatorSegment;

    {attribute 'pytmc' := 'pv: 25; link: 2550:'}
    fbSegment_25 : FB_UndulatorSegment;

    {attribute 'pytmc' := 'pv: 26; link: 2650:'}
    fbSegment_26 : FB_UndulatorSegment;

    {attribute 'pytmc' := 'pv: 27; link: 2750:'}
    fbSegment_27 : FB_UndulatorSegment;

    {attribute 'pytmc' := 'pv: 28; link: 2850:'}
    fbSegment_28 : FB_UndulatorSegment;

    {attribute 'pytmc' := 'pv: 29; link: 2950:'}
    fbSegment_29 : FB_UndulatorSegment;

    {attribute 'pytmc' := 'pv: 30; link: 3050:'}
    fbSegment_30 : FB_UndulatorSegment;

    {attribute 'pytmc' := 'pv: 31; link: 3150:'}
    fbSegment_31 : FB_UndulatorSegment;

    {attribute 'pytmc' := 'pv: 32; link: 3250:'}
    fbSegment_32 : FB_UndulatorSegment;

    {attribute 'pytmc' := 'pv: 33; link: 3350:'}
    fbSegment_33 : FB_UndulatorSegment;

    {attribute 'pytmc' := 'pv: 34; link: 3450:'}
    fbSegment_34 : FB_UndulatorSegment;

    {attribute 'pytmc' := 'pv: 36; link: 3650:'}
    fbSegment_36 : FB_UndulatorSegment;

    {attribute 'pytmc' := 'pv: 37; link: 3750:'}
    fbSegment_37 : FB_UndulatorSegment;

    {attribute 'pytmc' := 'pv: 38; link: 3850:'}
    fbSegment_38 : FB_UndulatorSegment;

    {attribute 'pytmc' := 'pv: 39; link: 3950:'}
    fbSegment_39 : FB_UndulatorSegment;

    {attribute 'pytmc' := 'pv: 40; link: 4050:'}
    fbSegment_40 : FB_UndulatorSegment;

    {attribute 'pytmc' := 'pv: 41; link: 4150:'}
    fbSegment_41 : FB_UndulatorSegment;

    {attribute 'pytmc' := 'pv: 42; link: 4250:'}
    fbSegment_42 : FB_UndulatorSegment;

    {attribute 'pytmc' := 'pv: 43; link: 4350:'}
    fbSegment_43 : FB_UndulatorSegment;

    {attribute 'pytmc' := 'pv: 44; link: 4450:'}
    fbSegment_44 : FB_UndulatorSegment;

    {attribute 'pytmc' := 'pv: 45; link: 4550:'}
    fbSegment_45 : FB_UndulatorSegment;

    {attribute 'pytmc' := 'pv: 46; link: 4650:'}
    fbSegment_46 : FB_UndulatorSegment;

    {attribute 'pytmc' := 'pv: 47; link: 4750:'}
    fbSegment_47 : FB_UndulatorSegment;



    fbSegment : ARRAY [iLowBound..iHighBound] OF POINTER TO FB_UndulatorSegment;
    fbCurrentSegment : REFERENCE TO FB_UndulatorSegment;

    iIndex : UDINT;

    bInitialized : BOOL := FALSE;

END_VAR

VAR CONSTANT
    {attribute 'pytmc' := '
        pv: FirstSegment
        io: i'}
    iLowBound  : UDINT := 21;
    {attribute 'pytmc' := '
        pv: LastSegment
         io: i'}
    iHighBound : UDINT := 47;
    {attribute 'pytmc' := '
        pv: Period_Short
        io: i
        field: EGU mm
    '}
    fPeriod_39_mm : LREAL := 39.0;

    {attribute 'pytmc' := '
        pv: Period_Long
        io: i
        field: EGU mm
    '}
    fPeriod_56_mm : LREAL := 56.0;

    {attribute 'pytmc' := '
        pv: LowK
        io: i
    '}
    fLowK : LREAL := 0.8;

    {attribute 'pytmc' := '
        pv: HiK
        io: i
    '}
    fHiK : LREAL := 5.7;
END_VAR



IF NOT bInitialized THEN
    Init();
END_IF

UndAdrUpdate();

nSeedUndulator := 0;
nTargetSeedUndulator := 0;

FOR iIndex := iLowBound TO iHighBound DO
    IF fbSegment[iIndex] <> 0 THEN
        fbCurrentSegment REF= fbSegment[iIndex]^;
        fbCurrentSegment(fbElectronEnergy:=fbElectronEnergy);
		fbCurrentSegment.fPeriod_mm := fbCurrentSegment.fLambda_U*1000;
		
        //Mark the seed undulator, first undulator operating within K bounds
        IF fbCurrentSegment.xActive AND nSeedUndulator = 0 THEN
            nSeedUndulator := iIndex;
            fCurrentPhotonEnergy := fbCurrentSegment.fPhotonEnergyAct;
        END_IF

        IF fbCurrentSegment.xTargetActive AND nTargetSeedUndulator = 0 THEN
            nTargetSeedUndulator := iIndex;
            fTargetPhotonEnergy := fbCurrentSegment.fPhotonEnergyDes;
        END_IF
    END_IF
END_FOR

IF nSeedUndulator = 0 THEN
    fCurrentPhotonEnergy := 0;
END_IF

IF nTargetSeedUndulator = 0 THEN
    fTargetPhotonEnergy := 0;
END_IF

ACTION Init:

UndAdrUpdate();

FOR iIndex := iLowBound TO iHighBound DO
        IF fbSegment[iIndex] <> 0 THEN
        fbCurrentSegment REF= fbSegment[iIndex]^;
        fbCurrentSegment.fLowK := fLowK;
        fbCurrentSegment.fHiK := fHiK;
    END_IF
END_FOR
bInitialized := TRUE;
END_ACTION

PROPERTY rCurrentPhotonEnergy : REAL
GET
rCurrentPhotonEnergy := fCurrentPhotonEnergy;
END_GET
END_PROPERTY

PROPERTY rTargetPhotonEnergy : REAL
GET
rTargetPhotonEnergy := fTargetPhotonEnergy;
END_GET
END_PROPERTY

ACTION UndAdrUpdate:
fbSegment[21] := 0;
fbSegment[22] := ADR(fbSegment_22);
fbSegment[23] := ADR(fbSegment_23);
fbSegment[24] := ADR(fbSegment_24);
fbSegment[25] := ADR(fbSegment_25);
fbSegment[26] := ADR(fbSegment_26);
fbSegment[27] := ADR(fbSegment_27);
fbSegment[28] := ADR(fbSegment_28);
fbSegment[29] := ADR(fbSegment_29);
fbSegment[30] := ADR(fbSegment_30);
fbSegment[31] := ADR(fbSegment_31);
fbSegment[32] := ADR(fbSegment_32);
fbSegment[33] := ADR(fbSegment_33);
fbSegment[34] := ADR(fbSegment_34);
fbSegment[35] := 0;
fbSegment[36] := ADR(fbSegment_36);
fbSegment[37] := ADR(fbSegment_37);
fbSegment[38] := ADR(fbSegment_38);
fbSegment[39] := ADR(fbSegment_39);
fbSegment[40] := ADR(fbSegment_40);
fbSegment[41] := ADR(fbSegment_41);
fbSegment[42] := ADR(fbSegment_42);
fbSegment[43] := ADR(fbSegment_43);
fbSegment[44] := ADR(fbSegment_44);
fbSegment[45] := ADR(fbSegment_45);
fbSegment[46] := ADR(fbSegment_46);
fbSegment[47] := ADR(fbSegment_47);
END_ACTION

END_FUNCTION_BLOCK

// MajorComponents/PhotonEnergyInterface/FB_LPhotonEnergy
FUNCTION_BLOCK FB_LPhotonEnergy EXTENDS FB_PhotonEnergy
VAR_INPUT
END_VAR
VAR_OUTPUT
END_VAR
VAR
    {attribute 'pytmc' := '
        pv: eEnrg
        link: BEND:DMPH:400:BACT
        field: EGU GeV
    '}
    fbHgvpuElectronEnergy : FB_LREALFromEPICS;

    {attribute 'pytmc' := '
        pv: EEnergy
        io: i
        field: DESC Electron Energy
        field: EGU GeV
    '}
    fElectronEnergyVal : LREAL;

    {attribute 'pytmc' := '
        pv: EEnergyValid
        io: i
        field: DESC Electron Energy Valid
    '}
    bElectronEnergyValid : BOOL;

    {attribute 'pytmc' := '
        pv: UND
        link: USEG:UNDH:
    '}
    fbHgvpu : FB_Hgvpu;

END_VAR

// Update PVs
fbHgvpuElectronEnergy();

fElectronEnergyVal := fbHgvpuElectronEnergy.fValue;
bElectronEnergyValid := fbHgvpuElectronEnergy.bValid;

fbHgvpu(fbElectronEnergy:=fbHgvpuElectronEnergy);

SUPER^(BP:=SUPER^.BP, Undulator:=fbHgvpu );

END_FUNCTION_BLOCK

// MajorComponents/PMPS_MPS_Interface/FB_BeamClassOutputs
(*
Sets the beam class assertion lines for a given beam class.
*)
{attribute 'no_check'}
FUNCTION_BLOCK FB_BeamClassOutputs
VAR_INPUT
    BP : ST_BeamParams;
END_VAR
VAR_OUTPUT
END_VAR
VAR
    nBeamClass   :    BYTE;
    wBeamClass    :    BYTE;

    InitCounter: BYTE;
    counter    :    INT;

    // Beam class lines are restricted to 8 channels in the current design, since
    // there are no plans to use all 16. Channels 1-7 may be allocated to any other
    // beam classes so long as they are ordered least to greatest.
    // Channel 8 is reserved for full beam.
    {attribute 'pytmc' := 'pv: BeamClassChannel
        io: i
        field: DESC Hardwire channel state'}
        epicsBitmap : WORD;

    {attribute 'TcLinkTo' := '[1] := TIIB[PMPS_Premp]^Channel 1^Output;
                              [2] := TIIB[PMPS_Premp]^Channel 2^Output;
                              [3] := TIIB[PMPS_Premp]^Channel 3^Output;
                              [4] := TIIB[PMPS_Premp]^Channel 4^Output;

                              [5] := TIIB[PMPS_Premp]^Channel 5^Output;
                              [6] := TIIB[PMPS_Premp]^Channel 6^Output;
                              [7] := TIIB[PMPS_Premp]^Channel 7^Output;
                              [8] := TIIB[PMPS_Premp]^Channel 8^Output;'} // 8 - Full beam
    q_BC_ASSERTION_LINES    AT    %Q*    : ARRAY [1..MAX_BEAM_CLASS_LINES] OF    BOOL;
END_VAR
VAR CONSTANT
    //Limited to total of 6 digital outputs
    MAX_BEAM_CLASS_LINES : BYTE := 8;
    BC_1HZ : BYTE := 1;
    BC_10HZ : BYTE := 2;
    BC_FULL : BYTE := 16;
END_VAR


// Determine BC
IF BP.nRate >= 120 THEN
    nBeamClass := BC_FULL;
ELSIF BP.nRate >= 10 THEN
    nBeamClass := BC_10HZ;
ELSIF BP.nRate >= 1 THEN
    nBeamClass := BC_1HZ;
ELSE
    nBeamClass := 0;
END_IF


//Assert Beam Class
////////////////////////////////////
//0x0 = 0000 0000 0000 0000
//0x1 = 0000 0000 0000 0001
//0xF = 1111 1111 1111 1111

//Initialize BC lines to zero on every pass
FOR InitCounter := 1 TO MAX_BEAM_CLASS_LINES DO
    q_BC_ASSERTION_LINES[InitCounter] := FALSE;
END_FOR

//Set BC lines according to beam class
//A BC of 0x0 would pass over this loop, setting none of the lines high
// , as FOR loops check the initialized variable at the top to see if it's >
// than the "TO" variable.
FOR wBeamClass:=1 TO MIN(MAX_BEAM_CLASS_LINES-1, nBeamClass) DO
    q_BC_ASSERTION_LINES[wBeamClass] := TRUE;
END_FOR

q_BC_ASSERTION_LINES[8] := nBeamClass = 16; //Set channel 8 true if BC is 16


// Readbacks for EPICS
epicsBitmap.0 := q_BC_ASSERTION_LINES[1];
epicsBitmap.1 := q_BC_ASSERTION_LINES[2];
epicsBitmap.2 := q_BC_ASSERTION_LINES[3];
epicsBitmap.3 := q_BC_ASSERTION_LINES[4];

epicsBitmap.4 := q_BC_ASSERTION_LINES[5];
epicsBitmap.5 := q_BC_ASSERTION_LINES[6];
epicsBitmap.6 := q_BC_ASSERTION_LINES[7];
epicsBitmap.7 := q_BC_ASSERTION_LINES[8];

END_FUNCTION_BLOCK

// MajorComponents/PMPS_MPS_Interface/FB_BeamClassOutputs_BCD
(*
Sets the beam class assertion lines for a given beam class.
*)
{attribute 'no_check'}
FUNCTION_BLOCK FB_BeamClassOutputs_BCD
VAR_INPUT
    BP : ST_BeamParams;
END_VAR
VAR_OUTPUT
END_VAR
VAR
    nBeamClass   :    BYTE;
    wBeamClass    :    BYTE;

    InitCounter: BYTE;
    counter    :    INT;

    // Beam class lines are restricted to 4 channels in the current design.
    // There are 16 possible beamclasses with 0 -15 with 0 no beam.
    // First out put is the LSB and bit 4 is MSB
    {attribute 'pytmc' := 'pv: BeamClassChannel
        io: i
        field: DESC Hardwire channel state'}
        epicsBitmap : WORD;

    {attribute 'TcLinkTo' := '[1] := TIIB[PMPS_Premp]^Channel 1^Output;
                              [2] := TIIB[PMPS_Premp]^Channel 2^Output;
                              [3] := TIIB[PMPS_Premp]^Channel 3^Output;
                              [4] := TIIB[PMPS_Premp]^Channel 4^Output;'}
    q_BC_ASSERTION_LINES    AT    %Q*    : ARRAY [1..MAX_BEAM_CLASS_LINES] OF    BOOL;
END_VAR
VAR CONSTANT
    //Limited to total of 4 digital outputs
    MAX_BEAM_CLASS_LINES : BYTE := 4;

END_VAR


//Initialize BC lines to zero on every pass
FOR InitCounter := 1 TO MAX_BEAM_CLASS_LINES DO
    q_BC_ASSERTION_LINES[InitCounter] := FALSE;
END_FOR

//Set BC lines according to beam class
// There are 4 digital outputs the BC is going to be a BCD
q_BC_ASSERTION_LINES[1] := BP.nBeamClass.0;
q_BC_ASSERTION_LINES[2] := BP.nBeamClass.1;
q_BC_ASSERTION_LINES[3] := BP.nBeamClass.2;
q_BC_ASSERTION_LINES[4] := BP.nBeamClass.3;

// Readbacks for EPICS
epicsBitmap.0 := q_BC_ASSERTION_LINES[1];
epicsBitmap.1 := q_BC_ASSERTION_LINES[2];
epicsBitmap.2 := q_BC_ASSERTION_LINES[3];
epicsBitmap.3 := q_BC_ASSERTION_LINES[4];

END_FUNCTION_BLOCK

// MajorComponents/PMPS_MPS_Interface/FB_BeamClassWatcher
(*
M. Ghaly
The Beam class watcher ensures the current and target beam class is within
the arbirated bounds.


The abritrated bounds come from a simple AND of all the permitted beam class ranges. See
the arbitrate action of the arbiter FB. It also reads a PV and ensures that the asserted Beam Class
is the same as the PV from the ATCA crate

Note, this protection logic does not account for beam-off when determining fast-fault
status. If a device is requesting a limited range of BC, this request must be honored,
regardless of current beam-rate.
*)
{attribute 'reflection'}
FUNCTION_BLOCK FB_BeamClassWatcher
VAR_INPUT
    i_stCurrentBeamParams    :    ST_BeamParams; //Link to global beam params
    i_stMachineTargetBeamParams    :    ST_BeamParams; //Link to global machine target beam params
    i_stRequestedBeamParams    :    ST_BeamParams; //Link to arbiter output or beam param. requestor
    //Auto Reset fault
    i_xAutoReset: BOOL;
    sName : STRING := 'BeamClassWatcher';
END_VAR
VAR_OUTPUT
END_VAR
VAR_IN_OUT
    io_fbFFHWO    :    FB_HardwareFFOutput;
END_VAR
VAR
    xBeamClassWithinBounds    :    BOOL;
    fbFF    :    FB_FastFault :=(
        i_DevName := sName,
        i_Desc := 'Fault occurs when the asserted beamclass or pv beam class falls outside the permitted range.',
        i_TypeCode := 7 );

   {attribute 'pytmc' := '
        pv: ResidualBeamClass
        io: i
        archive: 1Hz monitor
        field: EGU bc-bitmask
    '}
    bcResidual : DWORD;

    fbLog : FB_LogMessage := (
        eSubSystem := E_Subsystem.MPS,
        eSevr := TcEventSeverity.Critical
        );
    bLogOneShot : BOOL;
    sDevName : T_MaxString := 'Beam Class Watcher';

    fbGetHN : FB_GetHostName;
    bInit : BOOL := TRUE;

    {attribute 'instance-path'}
    {attribute 'noinit'}
    sPath    :    T_MaxString;

    fbStr : FB_FormatString := (
        sOut := 'Non-zero beam class residual: %32b; Req: %32b; Act: %32b');
END_VAR

IF bInit THEN
    fbGetHN(bExecute:=TRUE);
    bInit R= NOT fbGetHN.bBusy;
END_IF

xBeamClassWithinBounds := (i_stCurrentBeamParams.nBCRange AND i_stRequestedBeamParams.nBCRange) = i_stCurrentBeamParams.nBCRange
                    AND  (i_stCurrentBeamParams.nBeamClass <= i_stRequestedBeamParams.nBeamClass);

bcResidual := (i_stCurrentBeamParams.nBCRange XOR i_stRequestedBeamParams.nBCRange) AND i_stCurrentBeamParams.nBCRange;

IF bcResidual <> 0 AND bLogOneShot THEN
    fbLog.sJson := F_PMPS_JSON(
        CONCAT(fbGetHN.sHostName, sDevName),
        sPath,
        PMPS_CODES.PEW_FAULT);

    fbStr.arg1 := F_DWORD(bcResidual);
    fbStr.arg2 := F_WORD(i_stCurrentBeamParams.nBCRange);
    fbStr.arg3 := F_WORD(i_stRequestedBeamParams.nBCRange);

    fbStr();

    fbLog(sMsg:=fbStr.sOut);
    bLogOneShot := FALSE;
ELSIF bcResidual = 0 THEN
    bLogOneShot := TRUE;
END_IF

fbFF(i_xOK := xBeamClassWithinBounds OR (i_stCurrentBeamParams.nMachineMode = 0),
    io_fbFFHWO := io_fbFFHWO, i_xAutoReset := i_xAutoReset);

END_FUNCTION_BLOCK

// MajorComponents/PMPS_MPS_Interface/FB_CTLS_Outputs
(*
Controls auxiliary beam class outputs.

1-3 are mapped to control the Cu beamline rate via the LCLS II MPS.

Maps beam rate requests to 1, 10, or full rate beam for Cu linac.

*)
FUNCTION_BLOCK FB_CTLS_Outputs
VAR_INPUT
    BP    :    ST_BeamParams;
END_VAR
VAR_OUTPUT
END_VAR
VAR
    {attribute 'pytmc' := 'pv: CTLSChannel
        io: i
        field: DESC CTLS Rate Control hardwire channel state'}
    epicsBitmap : WORD;

    {attribute 'TcLinkTo' := '[1] := TIIB[PMPS_Premp]^Channel 9^Output;
                              [2] := TIIB[PMPS_Premp]^Channel 10^Output;
                              [3] := TIIB[PMPS_Premp]^Channel 11^Output;'}
    q_CLTS_ASSERTION_LINES    AT    %Q*    : ARRAY [1..3] OF    BOOL;



END_VAR


// CLTS 1Hz
q_CLTS_ASSERTION_LINES[1] := BP.nRate >= 1;
// CLTS 10Hz
q_CLTS_ASSERTION_LINES[2] := BP.nRate >= 10;
// CLTS Full rate
q_CLTS_ASSERTION_LINES[3] := BP.nRate >= 120;


epicsBitMap.0 := q_CLTS_ASSERTION_LINES[1];
epicsBitMap.1 := q_CLTS_ASSERTION_LINES[2];
epicsBitMap.2 := q_CLTS_ASSERTION_LINES[3];

END_FUNCTION_BLOCK

// MajorComponents/PMPS_MPS_Interface/FB_MachineModeFromEPICS
FUNCTION_BLOCK FB_MachineModeFromEPICS
(*
Readback options are:

0 – NC (normal conducting, copper linac)

1 – SC (superconducting linac)

2 – Misconfigured (something in link node not set correctly.

*)
VAR_IN_OUT
    BP : ST_BeamParams;
    fbMPS_MachineMode : FB_LREALFromEPICS;
    FFO : FB_HardwareFFOutput;
END_VAR
VAR_OUTPUT
    xError : BOOL;
END_VAR
VAR

    ffModeReadBack : FB_FastFault := (
        i_DevName := 'Arbiter',
        i_Desc := 'Issue with Machine mode readback from Accelerator. Gateway or EPICS connection. Must be fixed.',
        i_TypeCode := 16#313,
        i_xAutoReset:=True);
END_VAR
VAR CONSTANT
    cFailSafeMM : USINT := 3;
END_VAR

fbMPS_MachineMode();

IF fbMPS_MachineMode.bValid THEN
    BP.nMachineMode := LREAL_TO_USINT(fbMPS_MachineMode.fValue);
ELSE
    BP.nMachineMode := cFailSafeMM;
END_IF

ffModeReadBack(i_xOK:=(fbMPS_MachineMode.bValid) AND fbMPS_MachineMode.fValue <2 , io_fbFFHWO:=FFO);

BP.xValid R= NOT fbMPS_MachineMode.bValid;

END_FUNCTION_BLOCK

// MajorComponents/PMPS_MPS_Interface/FB_PhotonEnergyWatcher
(*
A. Wallace 2019-4-22
The photon energy watcher ensures the current and target photon energy is within
the arbirated bounds. Target in this case means, the calculated target photon energy
from the PVs that control the mechatronics of the undulators/ the electron energy.

If there are control PVs that match the monitor PVs, the control PVs are used to
calculate a "target" photon energy. This is supposed to cover when the undulators/
electron energy is transitioning.

The abritrated bounds come from a simple AND of all the permitted ranges. See
the arbitrate action of the arbiter FB.

Note, this protection logic does not account for beam-off when determining fast-fault
status. If a device is requesting a limited range of eV, this request must be honored,
regardless of current beam-rate.
*)
{attribute 'reflection'}
FUNCTION_BLOCK FB_PhotonEnergyWatcher
VAR_INPUT
    i_stCurrentBeamParams    :    ST_BeamParams; //Link to global beam params
    i_stMachineTargetBeamParams    :    ST_BeamParams; //Link to global machine target beam params
    i_stRequestedBeamParams    :    ST_BeamParams; //Link to arbiter output or beam param. requestor
    // Reset fault
    i_xReset: BOOL;
    sName : STRING := 'PhotonEnergyWatcher';
END_VAR
VAR_OUTPUT
END_VAR
VAR_IN_OUT
    io_fbFFHWO    :    FB_HardwareFFOutput;
END_VAR
VAR
    xPhotonEnergyWithinBounds    :    BOOL;
    fbFF    :    FB_FastFault :=(
        i_DevName := sName,
        i_Desc := 'Fault occurs when the calculated machine photon energy (K value calculated by undulator gap, and electron energy) falls outside the permitted range.',
        i_TypeCode := 7 );

   {attribute 'pytmc' := '
        pv: ResidualPhotonEnergies
        io: i
        archive: 1Hz monitor
        field: DESC Portions of beam eV not permitted
        field: EGU eV-bitmask
    '}
    evResidual : DWORD;

    fbLog : FB_LogMessage := (
        eSubSystem := E_Subsystem.MPS,
        eSevr := TcEventSeverity.Critical
        );
    bLogOneShot : BOOL;
    sDevName : T_MaxString := 'Photon Energy Watcher';

    fbGetHN : FB_GetHostName;
    bInit : BOOL := TRUE;

    {attribute 'instance-path'}
    {attribute 'noinit'}
    sPath    :    T_MaxString;

    fbStr : FB_FormatString := (
        sOut := 'Non-zero photon energy residual: %32b; Req: %32b; Act: %32b');
END_VAR

IF bInit THEN
    fbGetHN(bExecute:=TRUE);
    bInit R= NOT fbGetHN.bBusy;
END_IF

xPhotonEnergyWithinBounds := (i_stCurrentBeamParams.neVRange AND i_stRequestedBeamParams.neVRange) = i_stCurrentBeamParams.neVRange;

evResidual := (i_stCurrentBeamParams.neVRange XOR i_stRequestedBeamParams.neVRange) AND i_stCurrentBeamParams.neVRange;

IF evResidual <> 0 AND bLogOneShot THEN
    fbLog.sJson := F_PMPS_JSON(
        CONCAT(fbGetHN.sHostName, sDevName),
        sPath,
        PMPS_CODES.PEW_FAULT);

    fbStr.arg1 := F_DWORD(evResidual);
    fbStr.arg2 := F_DWORD(i_stCurrentBeamParams.neVRange);
    fbStr.arg3 := F_DWORD(i_stRequestedBeamParams.neVRange);

    fbStr();

    fbLog(sMsg:=fbStr.sOut);
    bLogOneShot := FALSE;
ELSIF evResidual = 0 THEN
    bLogOneShot := TRUE;
END_IF

fbFF(i_xOK := xPhotonEnergyWithinBounds,
    io_fbFFHWO := io_fbFFHWO,);

END_FUNCTION_BLOCK

// MajorComponents/SimulationFB/FB_eVSimulator
(* eV Simulator
A. Wallace 2019-8-30

Adds noise to the eV and changes eV position occasionally.
*)
FUNCTION_BLOCK FB_eVSimulator
VAR_INPUT
    NoiseLevel	:	REAL	:= 0; // eV Noise
    ChangeTime : TIME := T#10S;
END_VAR
VAR_OUTPUT
    eV	:	REAL := 300;
END_VAR
VAR
    eVRange : REAL := 1600;
    timer: TON;
    eVRand	:	DRAND :=(Seed:=0);
    NoiseRand : DRAND := (Seed:=0);
END_VAR


timer(in:=TRUE, PT:=ChangeTime);

//Occasionally change eV
IF timer.Q THEN
    timer(in:=FALSE);
    eVRand();
    eV := LIMIT(0, eVRange*LREAL_TO_REAL(eVRand.Num), eVRange);
END_IF

// Noise generation
NoiseRand();
eV := eV + NoiseLevel*LREAL_TO_REAL(NoiseRand.Num);
NoiseRand();
eV := LIMIT(0, ev - NoiseLevel*LREAL_TO_REAL(NoiseRand.Num), eVRange);

END_FUNCTION_BLOCK

// MajorComponents/SimulationFB/FB_MachineSimulator
(* Simulates the machine responding to requests by adding a bit of delay/ ramps
*)
FUNCTION_BLOCK FB_MachineSimulator
VAR_INPUT
    i_stAssertedParams    :    ST_BeamParams;
    i_xFault    :    BOOL;

    xEnableAtt : BOOL;
    xEnablePE : BOOL;
    xEnableRate : BOOL;
END_VAR
VAR_IN_OUT
    iq_stMachineParams    :    ST_BeamParams;
END_VAR
VAR
    nTargetTran: REAL;
    tonTranTimer    :    TON := (
        PT := T#2S
        );
    fTargetPP_mJ: REAL;
    tonPPETimer: TON := (
        PT := T#2S
    );
END_VAR


//Attenuation
IF xEnableAtt THEN
    IF i_stAssertedParams.nTran <> nTargetTran THEN
        tonTranTimer(IN:=FALSE);
        nTargetTran := i_stAssertedParams.nTran;
    ELSIF NOT tonTranTimer.Q THEN
        tonTranTimer(IN:=TRUE);
    ELSE
        iq_stMachineParams.nTran := nTargetTran;
    END_IF
END_IF

//Pulse Energy
(*
IF xEnablePE THEN
    IF i_stAssertedParams.fPP_mJ <> fTargetPP_mJ THEN
        tonPPETimer(IN:=FALSE);
        fTargetPP_mJ := i_stAssertedParams.fPP_mJ;
    ELSIF NOT tonTranTimer.Q THEN
        tonPPETimer(IN:=TRUE);
    ELSE
        iq_stMachineParams.fPP_mJ := fTargetPP_mJ;
    END_IF
END_IF
*)
//Rate
IF xEnableRate THEN
    IF i_xFault THEN
        iq_stMachineParams.nRate := 0;
    ELSE
        iq_stMachineParams.nRate := i_stAssertedParams.nRate;
    END_IF
END_IF

END_FUNCTION_BLOCK

// MajorComponents/Stoppers/FB_KStopper
FUNCTION_BLOCK FB_KStopper EXTENDS FB_StopperWatcher
VAR_INPUT
END_VAR
VAR_OUTPUT
END_VAR
VAR_IN_OUT
END_VAR
VAR
END_VAR

SUPER^(stCurrentBP:=SUPER^.stCurrentBP);

METHOD FB_init : BOOL
VAR_INPUT
    bInitRetains : BOOL; // if TRUE, the retain variables are initialized (warm start / cold start)
    bInCopyCode : BOOL;  // if TRUE, the instance afterwards gets moved into the copy code (online change)
    eStopper : K_Stopper;
    sStopperName : STRING;
END_VAR
Stopper := eStopper;
StopperName := sStopperName;
END_METHOD

END_FUNCTION_BLOCK

// MajorComponents/Stoppers/FB_StopperWatcher
// Relays stopper state and sends a message when stopper state changes.
FUNCTION_BLOCK FB_StopperWatcher
VAR_INPUT
END_VAR
VAR_OUTPUT
END_VAR
VAR_IN_OUT
    stCurrentBP : ST_BeamParams;
END_VAR
VAR
    i_StopperOutLS AT %I* : BOOL;
    i_StopperInLS AT %I* : BOOL;

    q_StopperOUT_Relay AT %Q* : BOOL;
    q_StopperIN_Relay AT %Q* : BOOL;

    Stopper : UINT;
    StopperName : STRING;
    {attribute 'instance-path'}
    {attribute 'noinit'}
    sPath    :    T_MaxString;

    // Logging
    fbLogMsg : FB_LogMessage := (
        eSubSystem := E_Subsystem.MPS);

    rtIn : R_TRIG;
    rtOut : R_TRIG;

    bInit: BOOL := TRUE;
END_VAR

IF bInit THEN
    fbLogMsg.sJson := F_PMPS_JSON(StopperName, sPath, 1000);
    bInit := FALSE;
END_IF


rtIn(CLK := i_StopperInLS);
rtOut(CLK := i_StopperOutLS);

IF rtIn.Q THEN
    fbLogMsg.sMsg := CONCAT(StopperName, ' moved IN');
    fbLogMsg();
ELSIF rtOut.Q THEN
    fbLogMsg.sMsg := CONCAT(StopperName, ' moved OUT');
    fbLogMsg();
END_IF

q_StopperOUT_Relay := i_StopperOutLS;
q_StopperIN_Relay := i_StopperInLS;

// Update current beam parameters
stCurrentBP.aVetoDevices[Stopper] := i_StopperInLS;

END_FUNCTION_BLOCK

// MajorComponents/Stoppers/FB_KVetoDevice
FUNCTION_BLOCK FB_KVetoDevice EXTENDS FB_VetoDevice
VAR_INPUT
END_VAR
VAR_OUTPUT
END_VAR
VAR
END_VAR

SUPER^(stCurrentBP:=SUPER^.stCurrentBP);

METHOD FB_init : BOOL
VAR_INPUT
    bInitRetains : BOOL; // if TRUE, the retain variables are initialized (warm start / cold start)
    bInCopyCode : BOOL;  // if TRUE, the instance afterwards gets moved into the copy code (online change)
    eVetoDeviceIN : K_Stopper := K_Stopper.DEFAULT;
    eVetoDeviceOUT : K_Stopper := K_Stopper.DEFAULT;
    sVetoDeviceName : STRING;
END_VAR
VetoDevice_IN := eVetoDeviceIN;
VetoDevice_OUT := eVetoDeviceOUT;
VetoDeviceName := sVetoDeviceName;
END_METHOD

END_FUNCTION_BLOCK

// MajorComponents/Stoppers/FB_VetoDevice
// Relays veto device state, updates current BP and sends a message when veto state changes.
FUNCTION_BLOCK FB_VetoDevice
VAR_INPUT
    i_bIn : BOOL;
    i_bOut : BOOL;
END_VAR
VAR_OUTPUT
    q_bIn : BOOL;
    q_bOut : BOOL;
END_VAR
VAR_IN_OUT
    stCurrentBP : ST_BeamParams;
END_VAR
VAR

    VetoDevice_IN : UINT := PMPS_GVL.MAX_VETO_DEVICES; // Veto device state array index
    VetoDevice_OUT : UINT := PMPS_GVL.MAX_VETO_DEVICES; // Veto device state array index

    VetoDeviceName : STRING;
    {attribute 'instance-path'}
    {attribute 'noinit'}
    sPath    :    T_MaxString;

    // Logging
        fbLogMsg : FB_LogMessage := (
            eSubSystem := E_Subsystem.MPS);

        rtIn : R_TRIG;
        rtOut : R_TRIG;
    ////////////////////////////////

    bInit: BOOL := TRUE;
END_VAR

IF bInit THEN
    fbLogMsg.sJson := F_PMPS_JSON(VetoDeviceName, sPath, 1000);
    bInit := FALSE;
END_IF

// Log
/////////////////////////////
    rtIn(CLK := i_bIn);
    rtOut(CLK := i_bOut);

    IF rtIn.Q THEN
        fbLogMsg.sMsg := CONCAT(VetoDeviceName, ' moved IN');
        fbLogMsg();
    ELSIF rtOut.Q THEN
        fbLogMsg.sMsg := CONCAT(VetoDeviceName, ' moved OUT');
        fbLogMsg();
    END_IF

// Relay
///////////////////////
    q_bIn := i_bIn;
    q_bOut := i_bOut;

// Update current beam parameters
/////////////////////////////////////
    stCurrentBP.aVetoDevices[VetoDevice_IN] := i_bIn;
    stCurrentBP.aVetoDevices[VetoDevice_OUT] := i_bOut;

END_FUNCTION_BLOCK

// MajorComponents/Stoppers/FB_LStopper
FUNCTION_BLOCK FB_LStopper EXTENDS FB_StopperWatcher
VAR_INPUT
END_VAR
VAR_OUTPUT
END_VAR
VAR_IN_OUT
END_VAR
VAR
END_VAR

SUPER^(stCurrentBP:=SUPER^.stCurrentBP);

METHOD FB_init : BOOL
VAR_INPUT
    bInitRetains : BOOL; // if TRUE, the retain variables are initialized (warm start / cold start)
    bInCopyCode : BOOL;  // if TRUE, the instance afterwards gets moved into the copy code (online change)
    eStopper : L_Stopper;
    sStopperName : STRING;
END_VAR
Stopper := eStopper;
StopperName := sStopperName;
END_METHOD

END_FUNCTION_BLOCK

// MajorComponents/Stoppers/FB_LVetoDevice
FUNCTION_BLOCK FB_LVetoDevice EXTENDS FB_VetoDevice
VAR_INPUT
END_VAR
VAR_OUTPUT
END_VAR
VAR
END_VAR

SUPER^(stCurrentBP:=SUPER^.stCurrentBP);

METHOD FB_init : BOOL
VAR_INPUT
    bInitRetains : BOOL; // if TRUE, the retain variables are initialized (warm start / cold start)
    bInCopyCode : BOOL;  // if TRUE, the instance afterwards gets moved into the copy code (online change)
    eVetoDeviceIN : L_Stopper := L_Stopper.DEFAULT;
    eVetoDeviceOUT : L_Stopper := L_Stopper.DEFAULT;
    sVetoDeviceName : STRING;
END_VAR
VetoDevice_IN := eVetoDeviceIN;
VetoDevice_OUT := eVetoDeviceOUT;
VetoDeviceName := sVetoDeviceName;
END_METHOD

END_FUNCTION_BLOCK

// MajorComponents/FB_BeamClassFromEPICS
FUNCTION_BLOCK FB_BeamClassFromEPICS

(*
enum MPSBeamClass {
    Beam Off    =  0,
    Kicker STBY =  1,
    BC1Hz       =  2,
    BC10Hz      =  3,
    Diagnostic  =  4,
    BC120Hz     =  5,
    Tuning      =  6,
    1% MAP      =  7,
    5% MAP      = 8,
    10% MAP     = 9,
    25% MAP     = 10,
    50% MAP     = 11,
    100% MAP    = 12,
    FULL        = 13,
    SPARE       = 14,
    SPARE       = 15
}
*)

VAR_IN_OUT
    BP : ST_BeamParams;
    fbMPS_BeamClass : FB_LREALFromEPICS;
    FFO : FB_HardwareFFOutput;
END_VAR
VAR_OUTPUT
    xError : BOOL;
END_VAR
VAR


    ffBeamClassReadBack : FB_FastFault := (
        i_DevName := 'Arbiter',
        i_Desc := 'Issue with beam class readback from Accelerator. Gateway or EPICS connection. Must be fixed.',
        i_TypeCode := 16#213,
        i_xAutoReset:=True);
END_VAR
VAR CONSTANT
    cFailSafeBC : USINT := 16;
END_VAR

fbMPS_BeamClass();

IF fbMPS_BeamClass.bValid THEN
    BP.nBeamClass := LREAL_TO_USINT(fbMPS_BeamClass.fValue);
ELSE
    BP.nBeamClass := cFailSafeBC;
END_IF
BP.nBCRange := TO_WORD(BP.nBeamClass);

ffBeamClassReadback(i_xOK:=fbMPS_BeamClass.bValid, io_fbFFHWO:=FFO);

BP.xValid R= NOT fbMPS_BeamClass.bValid;

END_FUNCTION_BLOCK

// MajorComponents/FB_BPControlDevice
(*
Used to request a beam parameter set from EPICS.

Technically just one of these is needed in the entire
PMPS for a line.

*)
FUNCTION_BLOCK FB_BPControlDevice
VAR_INPUT
        (*  Requested pre-optic attenuation %  *)
        {attribute 'pytmc' := 'pv: ReqBP:Transmission
            io: o
            field: HOPR 1;
            field: LOPR 0;
            field: PREC 2;
        '}
        nTran : REAL := PMPS_GVL.TRANS_SCALING_FACTOR;
        (* Pulse-rate *)
        {attribute 'pytmc' := 'pv: ReqBP:Rate
            io: o
            field: EGU Hz
        '}
        nRate : UDINT := 10;
        (* Photon energy ranges *)
        {attribute 'pytmc' := 'pv: ReqBP:PhotonEnergyRanges
            io: o
            field: EGU eV'}
        {attribute 'displaymode' := 'binary'}
        neVRange : DWORD := 4294967295;
        (* Beamclass ranges *)
         {attribute 'pytmc' := 'pv: ReqBP:BeamClassRanges
            io: o'}
        {attribute 'displaymode' := 'binary'}
        nBCRange : WORD := 32767;
END_VAR
VAR_OUTPUT
END_VAR
VAR_IN_OUT
    Arbiter : FB_Arbiter;
END_VAR
VAR
    EpicsReqBP : ST_BeamParams;
    {attribute 'pytmc' := '
        pv: ReqBP:Apply
        io: o
    '}
    bApply : BOOL;

    nControlDeviceID : DWORD;
    sControlDeviceName: STRING:= 'BP Control Device';
    rtApply : R_TRIG;

END_VAR


EpicsReqBP.nTran := nTran;
EpicsReqBP.neVRange := neVRange;
EpicsReqBP.nRate := nRate;
EpicsReqBP.nBCRange := nBCRange;

rtApply(CLK:=bApply);
IF rtApply.Q THEN
    Arbiter.RemoveRequest(nControlDeviceID);
    Arbiter.AddRequest(nControlDeviceID, EpicsReqBP, sControlDeviceName);
    bApply := FALSE;
END_IF

METHOD FB_init : BOOL
VAR_INPUT
    bInitRetains : BOOL; // if TRUE, the retain variables are initialized (warm start / cold start)
    bInCopyCode : BOOL;  // if TRUE, the instance afterwards gets moved into the copy code (online change)
    nID : DWORD := PMPS_GVL.EXCLUDED_ASSERTION_ID;
END_VAR
nControlDeviceID:= nID;
END_METHOD

END_FUNCTION_BLOCK

// MajorComponents/FB_BPRequestor
(* BP Requestor
Elevates the BP request from an arbiter to PMPS_GVL.stRequestedBP
*)
FUNCTION_BLOCK FB_BPRequestor IMPLEMENTS I_HigherAuthority
VAR_INPUT
END_VAR
VAR_OUTPUT
    q_ReqBP : ST_BeamParams; // Arbitrated BP
END_VAR
VAR_IN_OUT
    Arbiter : FB_Arbiter;
    //FFO : FB_HardwareFFOutput;
END_VAR
VAR
    ReqBP : ST_BeamParams;
    nCohort : ULINT; // Current cohort, inc. 1 cycle after IO is updated
    nRequestCohort : ULINT; // Cohort number recorded at the time of the request.
END_VAR

Arbiter.ElevateRequest(THIS^); // Executes arbitration and retrieves ReqBP

IF nRequestCohort >= nCohort THEN
    // Update requested BP set
    q_ReqBP := ReqBP;
    // Note: we may do more here someday... perhaps all of the output control
    // will reside in here, and be solely controlled by this block. For now
    // I am going to adopt a flat management structure.
    // Start a new cohort
    nCohort := nCohort + 1;
END_IF

// Returns true when outputs to MPS are updated
METHOD CheckRequest : BOOL
VAR_INPUT
    nReqID	: DWORD;
END_VAR
VAR_INST
    xFirstTime : BOOL;
    nId : DWORD;
END_VAR
(* nRequestCohort will be < nCohort after output control
function blocks have been updated to reflect the new request
*)
CheckRequest := nRequestCohort < nCohort;
END_METHOD

METHOD RemoveRequest : BOOL
VAR_INPUT
    nReqID    :    DWORD; //StateID to remove
END_VAR
END_METHOD

METHOD RequestBP : BOOL
VAR_INPUT
    (*StateID of state requesting beam parameter set*)
    nReqID	: DWORD;
    (*Requested beam params*)
    stReqBP	: ST_BeamParams;
END_VAR
VAR_INST
    ReqID : DWORD;
    Registered : BOOL := FALSE;
END_VAR

// Check the request is coming from the same source we're used to
IF NOT Registered THEN
    ReqID := nReqID;
    Registered := TRUE;
END_IF
// log a complaint if false
RequestBP := ReqId = nReqId;

// Update internal BP request struct
ReqBP := stReqBP;

// Record current cohort

    nRequestCohort := nCohort;
END_METHOD

END_FUNCTION_BLOCK

// MajorComponents/FB_LinearGovernor

(* The governor is meant to check your work and keep you from making mistakes.

Checks:
Does your state match the device position and visa versa?
Are the beam parameters safe for the device state?
Did you properly assert the transition and final beam parameters?

*)
FUNCTION_BLOCK FB_LinearGovernor
VAR_INPUT
    i_stCurrentBeamParams    :    ST_BeamParams; //Link to global beam params
    i_xMPSOverride            :    BOOL; //True releases MPS limits after a delay
    i_xTransitionRequested    :    BOOL; //Set true to request a transition
    i_xResetMPSFault    :    BOOL; //Set true to clear MPS fault
END_VAR
VAR_OUTPUT
     //True when governor has released restrictions
    q_xTransitionPermitted    :    BOOL;
    //Set if MC_Power has an error, or override mode is requested
    q_xFault    :    BOOL;
    // Indicates override mode is active
    q_xMPSLimitsOverridden: BOOL;
END_VAR
VAR_IN_OUT
    stDevice    :    ST_Device; //The governed
    Arbiter    :    FB_Arbiter;
    FastFaultOutput    :    FB_HardwareFFOutput;
END_VAR
VAR
    mcPower    :    MC_Power;

    xActuatorPositiveEnable: BOOL;
    xActuatorNegativeEnable: BOOL;

    xMPSPositiveEnable    :    BOOL;
    xMPSNegativeEnable    :    BOOL;
    lrPosition: LREAL;

    lrLatchedTargetPosition    :    LREAL;
    lrLatchedTargetTolerance    :    LREAL;
    stLatchedTargetState    :    ST_DeviceStateExt;

    lrMPSUpperLimit: LREAL;
    lrMPSLowerLimit: LREAL;
    rtNewState: R_TRIG;
    xTransitionOK: BOOL;

    tonMPSOverrideMode    :    TON := (
        PT := T#5S
    );

    srMPSFault    :    SR;
    // Actuator out of bounds fault
    xActuatorOOB: BOOL;
    //Beam parameters out of spec
    xBeamParamsOOS: BOOL;
    //Beam parameters of currently latched state

    stLatchedBeamParams: ST_BeamParams;
    stTargetState: ST_DeviceStateExt;

    rtLatchNewState    :    R_TRIG;
    xInit: BOOL := TRUE;

    stInitDeviceState: ST_DeviceStateExt;
    // Indicates an error with initialization
    xInitFault: BOOL;
    // Indicates the state could not be found in the state table. There may be something wrong in the device state machine implementation or state table instantiation.
    xStateLookupError: BOOL;
    // A transition needs to be requested at least once before we start latching any state.
    xTransitionHasBeenRequested: BOOL := FALSE;
    ffBeamParamsOK : FB_FastFault;
    ffActuatorBoundsOK    :    FB_FastFault;
END_VAR


lrPosition := stDevice.stAxis.NcToPlc.ActPos; //Actuator position

stDevice.stAxis.ReadStatus();
//Init
(* The init strategy is:
If the device is restored and it's residing at the safe position,
no PMPS faults. *)
////////////////////////////////
    IF xInit THEN
        xInit := FALSE;
        //Use nSafeSate for initialization.
        stDevice.StateTable.A_Lookup(key := stDevice.nSafeState);
        IF stDevice.StateTable.bOk THEN
            stInitDeviceState := F_DeviceState_To_DeviceStateExt(stDevice.StateTable.getValue, TRUE);
            xInitFault := FALSE;
        ELSE
            xInitFault := TRUE;
            stInitDeviceState.xValid := FALSE;
        END_IF
        lrLatchedTargetPosition := stInitDeviceState.rPosition;
        lrLatchedTargetTolerance := stInitDeviceState.rTolerance;
        stLatchedBeamParams := stInitDeviceState.stReqBeamParam;
    END_IF

// The governor will permit transitions once it verifies the transition assertion is active
// Note the governor does not verify the target state beam params are asserted, perhaps it should <TODO>
////////////////////////////////
    IF i_xTransitionRequested THEN
        xTransitionHasBeenRequested    := TRUE;

        xTransitionOK := Arbiter.CheckRequest( stDevice.stTransitionState.nStateRef) AND F_SafeBPCompare(i_stCurrentBeamParams, stDevice.stTransitionState.stReqBeamParam);

        //Set the target state for evaluation in further logic
        stdevice.StateTable.A_Lookup(key := stDevice.nTargetState);
        IF stDevice.StateTable.bOk THEN
            stTargetState := F_DeviceState_To_DeviceStateExt(stDevice.StateTable.getValue, TRUE);
            xStateLookupError := FALSE;
        ELSE
            xStateLookupError := TRUE;
            stTargetState.xValid := FALSE;
        END_IF
    ELSE
        xTransitionOK := FALSE;
    END_IF

(* Note about TransitionRequested

If TransitionRequested goes false during a transition, an MPS fault may be induced. This occurs
because the Actuator Out of Bounds fault will go back to using the original state limits, which
the axis may have already moved beyond.

To avoid this transient fault, make sure your device state machine is implemented such that the
transition request to the governor block remains high until the target position is reached.
*)

//Determine if a transition is complete and latch the new state
(* A transition is complete when:

Axis at standstill.
Axis within tolerance.
No transition req.

Once these conditions are met, the MPS limits shall re-engage to restrict the
axis motion to the tolerance around the state position and the MPS fault monitors
shall evaluate based on the newly latched target state.
*)

rtLatchNewState(CLK := stDevice.stAxis.Status.StandStill AND
    lrPosition <= stTargetState.rPosition + stTargetState.rTolerance AND
    lrPosition >= stTargetState.rPosition - stTargetState.rTolerance AND
    NOT i_xTransitionRequested AND xTransitionHasBeenRequested);

IF rtLatchNewState.Q THEN
    lrLatchedTargetPosition := stTargetState.rPosition;
    lrLatchedTargetTolerance := stTargetState.rTolerance;
    stLatchedBeamParams := stTargetState.stReqBeamParam;
    stLatchedTargetState := stTargetState;
END_IF

//Let other blocks know the governor won't interfer with transitions
q_xTransitionPermitted := xTransitionOK;

//Adjust limit ranges based on active state and current target
IF xTransitionOK THEN
    //Extend range to include target state
    lrMPSUpperLimit := MAX(lrMPSUpperLimit, stTargetState.rPosition + stTargetState.rTolerance);
    lrMPSLowerLimit := MIN(lrMPSLowerLimit, stTargetState.rPosition - stTargetState.rTolerance);
ELSE
    //Calculate the limit positions for MPS based on current state
    lrMPSUpperLimit := lrLatchedTargetPosition + lrLatchedTargetTolerance;
    lrMPSLowerLimit := lrLatchedTargetPosition - lrLatchedTargetTolerance;
END_IF


//MPS override
(* In override mode, the device will be free to move anywhere within it's travel range *)
//Permit motion after a small delay
tonMPSOverrideMode(IN:=i_xMPSOverride OR stDevice.xOverrideMPSLimits, Q=>q_xMPSLimitsOverridden);

//Virtual limit switch evaluation
xActuatorPositiveEnable    := stDevice.i_xHiLim AND lrPosition <= stDevice.lrUpperPositionLimit;
xActuatorNegativeEnable    := stDevice.i_xLoLim AND lrPosition >= stDevice.lrLowerPositionLimit;

//Evaluate MPS limit states
xMPSPositiveEnable := lrPosition <= lrMPSUpperLimit;
xMPSNegativeEnable := lrPosition >= lrMPSLowerLimit;

//Final Limit switch evaluation
mcPower.Enable_Positive := xActuatorPositiveEnable AND (tonMPSOverrideMode.Q OR xMPSPositiveEnable);
mcPower.Enable_Negative := xActuatorNegativeEnable AND (tonMPSOverrideMode.Q OR xMPSNegativeEnable);

mcPower(
    Axis := stDevice.stAxis,
    Enable := stDevice.xEnable //link to device enable <TODO>
);



//MPS Faults
//Fault if the beam is unsafe for current state
ffBeamParamsOK(i_xOK:=F_SafeBPCompare(i_stCurrentBeamParams, stLatchedBeamParams),
                i_xReset:=i_xResetMPSFault,
                io_fbFFHWO := FastFaultOutput);

//Fault if the position is outside of the permitted range
ffActuatorBoundsOK(i_xOK := (lrPosition <= lrMPSUpperLimit AND lrPosition >= lrMPSLowerLimit),
                    i_xReset:=i_xResetMPSFault,
                io_fbFFHWO := FastFaultOutput);



//Collect all other faults
q_xFault := NOT ffBeamParamsOK.o_xFFLine OR
    NOT ffActuatorBoundsOK.o_xFFLine OR
    mcPower.Error    OR
    i_xMPSOverride    OR
    xInitFault;

//Any faults trip the fast fault line for this FB
//FastFaultOutput.CheckIn(NOT q_xFault);

END_FUNCTION_BLOCK

// MajorComponents/FB_RateFromEPICS
FUNCTION_BLOCK FB_RateFromEPICS

(*
enum MPSBeamRates {
    MPSRateInvalid            =  0,
    MPSRate0Hz                =  1,
    /* Previously used 2 and 3 for single shot and burst */
    MPSRate1Hz                =  4,
    MPSRate10Hz               =  5,
    MPSRate30Hz               =  6,
    MPSRate60Hz               =  7,
    MPSRate120Hz              =  8,
    MPSRateUnknown            =  9,
    MPSRateSingleShot         = 10,
    MPSRateBurstMode          = 11,
    MPSRateBurstModeNotActive = 12,
    MPSNumberOfBeamRates      = 13,
    MPSRateBurstInvalid       = 14
}
*)

VAR_IN_OUT
    BP : ST_BeamParams;
    fbBYKIK_Rate : FB_LREALFromEPICS;
    FFO : FB_HardwareFFOutput;
END_VAR
VAR_OUTPUT
    xError : BOOL;
END_VAR
VAR


    eMPSRate : E_MPSBeamRates;

    ffRateReadBack : FB_FastFault := (
        i_DevName := 'Arbiter',
        i_Desc := 'Issue with rate readback from Accelerator. Gateway or EPICS connection. Must be fixed.',
        i_TypeCode := 16#203,
        i_xAutoReset:=True);
END_VAR
VAR CONSTANT
    cFailSafeRate : UDINT := 1000001;
END_VAR

fbBYKIK_Rate();

IF fbBYKIK_Rate.bValid THEN
    eMPSRate := LREAL_TO_UINT(fbBYKIK_Rate.fValue);
ELSE
    eMPSRate := E_MPSBeamRates.MPSRateInvalid;
END_IF

CASE eMPSRate OF
    MPSRateInvalid:
        BP.nRate := cFailSafeRate;
    MPSRate0Hz:
        BP.nRate := 0;
    MPSRate1Hz:
        BP.nRate := 1;
    MPSRate10Hz:
        BP.nRate := 10;
    MPSRate30Hz:
        BP.nRate := 30;
    MPSRate60Hz:
        BP.nRate := 60;
    MPSRate120Hz:
        BP.nRate := 120;
    MPSRateUnknown:
        BP.nRate := cFailSafeRate;

ELSE
    BP.nRate := cFailSafeRate;
END_CASE

ffRateReadback(i_xOK:=fbBYKIK_Rate.bValid, io_fbFFHWO:=FFO);

BP.xValid R= NOT fbBYKIK_Rate.bValid OR
            eMPSRate = MPSRateUnknown OR
            eMPSRate = MPSRateInvalid;

END_FUNCTION_BLOCK

// TestComponents/FB_Arbiter_Test
{attribute 'call_after_init'}
FUNCTION_BLOCK FB_Arbiter_Test EXTENDS TcUnit.FB_TestSuite
VAR_INPUT
END_VAR
VAR_OUTPUT
END_VAR
VAR
END_VAR

Arbitration();
RequestCheckRemoveBP();
FullArbitrationStack();
StackArbiters();
RemoveReq();
DoS();

METHOD ArbiterCapacity
VAR_INPUT
END_VAR
VAR
    nId    :    DWORD := 1;
    stReq    :    ST_BeamParams := (nTran:=12);

    nRandID : DWORD;
    testReq : ST_BeamParams := (neVRange := 16#FFEE, nRate:=33);

    idx : DWORD;

END_VAR
VAR_INST
    fbArbCapacityTest    :    FB_Arbiter(1);

    Cycle : INT := 0;

    CycleLimit : INT := 20;

END_VAR
VAR CONSTANT
    SysID : DWORD := 42;
END_VAR

TEST('Arbiter Capcity');
    // Fill the arbiter
    FOR idx := 1 TO PMPS_PARAM.MAX_ASSERTIONS DO
        fbArbCapacityTest.AddRequest(nReqID := idx, stReqBP := testReq, sDevName:= CONCAT('Device #', TO_STRING(idx)));
    END_FOR

TEST_FINISHED();
END_METHOD

METHOD Arbitration
VAR_INPUT
END_VAR
VAR

     nTranReqID    :    UDINT    := 1;
    stAttReqBP    :    ST_BeamParams := PMPS_GVL.cstFullBeam;

    nPPEReqID    :    UDINT    := 2;
    stPPEReqBP    :    ST_BeamParams := PMPS_GVL.cstFullBeam;

    nEVReqID    :    UDINT    := 3;
    stEVReqBP    :    ST_BeamParams := PMPS_GVL.cstFullBeam;

    nRateReqID    :    UDINT    := 4;
    stRateReqBP    :    ST_BeamParams := PMPS_GVL.cstFullBeam;

    nBCRangeReqID : UDINT    := 5;
    stBCReqBP    :    ST_BeamParams := PMPS_GVL.cstFullBeam;

    stArbitratedBP    :    ST_BeamParams;// :=  PMPS_GVL.cstFullBeam;;
    stExpectedBP    :    ST_BeamParams := PMPS_GVL.cstFullBeam;

END_VAR
VAR_INST
    fbArbiter    :    FB_Arbiter(1);
END_VAR
TEST('Arbitration');

stAttReqBP.nTran := 0.50;
stEVReqBP.neVRange := 2#1111_1111_1111_1111_1111_1100_1111_1111;
stRateReqBP.nRate := 10;
stBCReqBP.nBCRange := 2#0111_0000_0000_0000;
stBCReqBP.nBeamClass := 15;

stExpectedBP.nTran     := stAttReqBP.nTran;
stExpectedBP.neVRange := stEVReqBP.neVRange;
stExpectedBP.nRate := stRateReqBP.nRate;
stExpectedBP.nBCRange := stBCReqBP.nBCRange;
stExpectedBP.nBeamClass := stBCReqBP.nBeamClass;


//Load arbiter with beam parameter sets
AssertTrue(fbArbiter.AddRequest(nTranReqID, stAttReqBP, sDevName:= 'Device' ),
                    'Safest attenuation request failed to load');

//Load arbiter with beam parameter sets
AssertTrue(fbArbiter.AddRequest(nPPEReqID, stPPEReqBP, sDevName:= 'Device'),
                    'Safest PPE request failed to load');

